VAR
	iter : FB_ObjCollectIterator;
END_VAR
//Bei dieser Methode wird der Node nur auf der Collection entnommen aber nicht gelöscht.
//Wird nur genutzt, wenn sich die Position eines Nodes im Object-Tree ändert (ExchangePiece)
IF pNode > 0 AND_THEN pNode^.nodes.nCount = 0 THEN
	M_GetIterator(iter);
	WHILE iter.pNode > 0 DO
		IF pNode = iter.pNode THEN
			IF pNode = pHead THEN
				pHead := pHead^.pNext;
				IF pHead > 0 THEN
					pHead^.pPrev := 0;	
				END_IF
			ELSIF pNode = pTail THEN
				pTail := pTail^.pPrev;
				IF pTail > 0 THEN
					pTail^.pNext := 0;	
				END_IF
			ELSE
				pNode^.pPrev^.pNext := pNode^.pNext;
				pNode^.pNext^.pPrev := pNode^.pPrev;
			END_IF
			pNode^.P_pOwnerColl := 0;
			nCount := nCount - 1;
			EXIT;
		END_IF
		iter.M_Increment();
	END_WHILE
END_IF
END_METHOD

END_FUNCTION_BLOCK

// ---- Configuration/FB_ObjCollectIterator.TcPOU
FUNCTION_BLOCK FB_ObjCollectIterator
VAR_INPUT
	pInitNode : POINTER TO FB_ObjCollectionNode;
END_VAR
VAR_OUTPUT
	pNode : POINTER TO FB_ObjCollectionNode;
END_VAR
VAR
END_VAR

pNode := pInitNode;

METHOD M_Increment
VAR_INPUT
END_VAR
IF pNode > 0 AND_THEN pNode^.pNext > 0 THEN
	pNode := pNode^.pNext;
ELSE
	pNode := 0;
END_IF
END_METHOD

END_FUNCTION_BLOCK

// ---- Configuration/FB_ObjCollectIteratorDeep.TcPOU
FUNCTION_BLOCK FB_ObjCollectIteratorDeep EXTENDS FB_ObjCollectIterator
VAR_INPUT
END_VAR
VAR_OUTPUT
END_VAR
VAR
	bBeforeInChild : BOOL;
	nLevel : UINT;
END_VAR

pNode := pInitNode;

METHOD M_Increment
VAR_INPUT
END_VAR

VAR
	
END_VAR
//Den kompletten Tree traversieren
//am Anfang steht der Iter auf dem Head von Level0
//wenn aktueller Node Childs hat, dann von diesen Childs neuen Iterator holen
//das geht immer so weiter bis ein Node keinen Child mehr hat
//wenn das eintritt, dann wird nach Nachbarn gesucht
//wenn ein Nachbar vorhanden, dann wird dieser zurückgegeben
//wenn kein Nachbar vorhanden, dann wird Parent zurückgegeben, hier besteht allerdings das Problem, dass
//wenn dann wieder inkrementiert wird, das Parent ja wieder auf das Child zugreifen würde. Ein Flag welches anzeigt,
//dass vorher schon in einer höheren Ebene dieses Parents gesucht wurde, könnte das lösen. Dieses muss allerdings immer
//an der richtigen stelle zurückgesetzt werden

IF pNode > 0 THEN
	IF pNode^.nodes.nCount > 0 THEN
		IF bBeforeInChild THEN
			//Nachbar suchen
			IF pNode^.pNext > 0 THEN
				pNode := pNode^.pNext;
			ELSE
				//kein Nachbar gefunden
				IF pNode^.pOwnerColl^.pOwnerNode > 0 THEN
					IF nLevel = 0 THEN
						pNode := 0;
						bBeforeInChild := FALSE;		
					ELSE
						//hier wird eine Ebene zurückgesprungen -> Flag setzen
						pNode := pNode^.pOwnerColl^.pOwnerNode;
						bBeforeInChild := TRUE;
						nLevel := nLevel - 1;
						THIS^.M_Increment();
					END_IF
				ELSE
					pNode := 0;
					bBeforeInChild := FALSE;		
				END_IF
			END_IF
			bBeforeInChild := FALSE;
		ELSE
			//Iterator vom neuen Child holen
			pNode^.nodes.M_GetIterator(THIS^);	//Hier wir das Level inkrementiert
			nLevel := nLevel + 1;
		END_IF
	ELSIF pNode^.pNext > 0 THEN
		//nach Nachbar suchen
		pNode := pNode^.pNext;
	ELSIF pNode^.pOwnerColl^.pOwnerNode > 0 AND nLevel > 0 THEN
		//hier wird eine Ebene zurückgesprungen -> Flag setzen
		pNode := pNode^.pOwnerColl^.pOwnerNode;
		bBeforeInChild := TRUE;
		nLevel := nLevel - 1;
		THIS^.M_Increment();
	ELSE
		pNode := 0;
		bBeforeInChild := FALSE;
	END_IF
END_IF
END_METHOD

END_FUNCTION_BLOCK

// ---- Objects/FB_Slot.TcPOU
{attribute 'enable_dynamic_creation'}
FUNCTION_BLOCK FB_Slot
VAR_INPUT
END_VAR
VAR_OUTPUT
END_VAR
VAR
	pOwner	: POINTER TO FB_Object;
	pChild	: POINTER TO FB_Object;
	nNr		: UINT;
	stRelPos: ST_3DPoint;
END_VAR

METHOD FB_init : BOOL
VAR_INPUT
	bInitRetains : BOOL; // if TRUE, the retain variables are initialized (warm start / cold start)
	bInCopyCode : BOOL;  // if TRUE, the instance afterwards gets moved into the copy code (online change)
	pOwner		: POINTER TO FB_Object;
END_VAR
THIS^.pOwner := pOwner;
END_METHOD

PROPERTY P_nNr : UINT
GET
P_nNr := nNr;
END_GET
SET
nNr := P_nNr;
END_SET
END_PROPERTY

PROPERTY P_rRelPosY : REAL
SET
stRelPos.Y := P_rRelPosY;
END_SET
GET
P_rRelPosY := stRelPos.Y;
END_GET
END_PROPERTY

PROPERTY P_rRelPosX : REAL
SET
stRelPos.X := P_rRelPosX;
END_SET
GET
P_rRelPosX := stRelPos.X;
END_GET
END_PROPERTY

PROPERTY P_pChild : POINTER TO FB_Object
GET
P_pChild := pChild;
END_GET
SET
pChild := P_pChild;
END_SET
END_PROPERTY

PROPERTY P_stRelPos : ST_3DPoint
SET
stRelPos := P_stRelPos;
END_SET
GET
P_stRelPos := stRelPos;
END_GET
END_PROPERTY

PROPERTY P_stAbsPos : ST_3DPoint
GET
VAR
	stTemp : ST_3DPoint;
	pMzTool: POINTER TO FB_MzTool;
	pTarget: POINTER TO FB_TargetBase;
END_VAR
IF pOwner^.P_eObjectType = E_ObjectType.OBJECTTYPE_MZHead THEN
	pMzTool := pOwner;
	stTemp := pMzTool^.P_stAbsPosTotal;
	stTemp.X := stTemp.X + stRelPos.X;
	stTemp.Y := stTemp.Y + stRelPos.Y;
	P_stAbsPos := stTemp;
ELSIF pOwner^.M_bIsGroup(E_ObjectGroup.OBJECTGROUP_MzTool) THEN
	pMzTool := pOwner;
	P_stAbsPos := F_Add3DPoints(stRelPos, pMzTool^.P_stAbsPosPhysExclPiece);
ELSIF pOwner^.M_bIsGroup(E_ObjectGroup.OBJECTGROUP_Target) THEN
	pTarget := pOwner;
	P_stAbsPos := F_Add3DPoints(stRelPos, pTarget^.P_stAbsPosLB);
END_IF
END_GET
END_PROPERTY

PROPERTY P_rRelPosZ : REAL
GET
P_rRelPosZ := stRelPos.Z;
END_GET
SET
stRelPos.Z := P_rRelPosZ;
END_SET
END_PROPERTY

END_FUNCTION_BLOCK

// ---- Objects/Tools/FB_MzTool.TcPOU
FUNCTION_BLOCK FB_MzTool EXTENDS FB_MzBase
VAR_INPUT
END_VAR
VAR_OUTPUT
END_VAR
VAR
	pParentMzTool		: POINTER TO FB_MzBase;
	
	nParentSlotNr		: UINT;	//LÖSCHEN!!!!!!!!!!!!!!!
	pZAxisRef 			: POINTER TO FB_ZAxisRef;
	pCurrentTarget		: POINTER TO FB_TargetBase;
	
	bIsMESTool			: BOOL;
	
	//Action: "JogZ"
	bJogZ				: BOOL;
	nStateA_JogZ		: USINT;			//State von A_Jog()
	fbZmJog				: FB_ZM_Jog;
	eJogZDirectionNew	: E_MoveDirection;
	eJogZDirection		: E_MoveDirection;
	bJogZForward		: BOOL;
	bJogZBackwards		: BOOL;
	bJogZClock			: BOOL;
	bJogZModeInchingNew	: BOOL;				//wenn True dann Tipbetrieb sonst kontinuierlich
	bJogZModeInching	: BOOL;				//wenn True dann Tipbetrieb sonst kontinuierlich
	rJogZDistance		: REAL;
	rJogZSpeed			: REAL;
	bJogZImpuls			: BOOL;
	
	//Ergänzung zu Action: MoveZ"
	nReducedMoveZSpeed	: DINT;
	nReducedMoveZDist	: DINT;
	
END_VAR

IF eCurrentState = E_MachineState.MACHINESTATE_Active THEN
	//BasicActions ausführen
	IF bJogZ THEN
		A_JogZ();
		IF nStateA_JogZ >= 80 THEN
			IF nStateA_JogZ >= 99 THEN
				bStopAllOnError := TRUE;
				bError := TRUE;
			END_IF
		bJogZ := FALSE;
		nStateA_JogZ := 0; 
		M_RemoveListEntry(nSearchValue:= E_Action.ACTION_Jog);
		END_IF
	END_IF
END_IF


SUPER^();	//FB_MzBase() aufrufen

//Prozessdaten aktualisieren
IF pZAxisRef > 0 THEN
	stProcessData.n32Data[3] := REAL_TO_DINT(pZAxisRef^.P_rCurrentPos);
END_IF
stCurrentPos := P_stCurrentPosTotal;
stProcessData.n32Data[4] := REAL_TO_DINT(stCurrentPos.X);
stProcessData.n32Data[5] := REAL_TO_DINT(stCurrentPos.Y);
stProcessData.n32Data[6] := REAL_TO_DINT(stCurrentPos.Z);

ACTION A_Init:
	IF nStateA_InitAxis = 0 THEN
		bInitAxisOk := FALSE;
		//Ist Z-Achse physikalisch vorhanden?
		IF NOT pZAxisRef^.stInput.nStatus.7 THEN
			stError.ErrorId := E_ErrorIdMultiZ.ERRORID_NoZAxis;
			stError.HardwareGrp := E_HardwareGrp.AxisZ;
			stError.HardwareNr	:= pZAxisRef^.nChannel;
			stError.POUState := nStateA_InitAxis;
			nStateA_InitAxis := 99;
		ELSE
			IF pZAxisRef^.stStatus.bIsHoming THEN //Homing dieser Achse wurde bereits durch ein anderes Tool oder Head angestoßen
				nStateA_InitAxis := 2;
			ELSE
				nStateA_InitAxis := 1;
			END_IF		
		END_IF
	END_IF
	
	IF nStateA_InitAxis = 1 THEN
		fbZmHome(bExecute:= TRUE, pFbZAxisRef:= pZAxisRef, bMoveToHome:= TRUE);
		P_bZIsMoving := TRUE;
		pParentMzTool^.P_bZIsMoving := TRUE;		
		IF NOT fbZmHome.bBusy THEN
			IF fbZmHome.bError THEN
				stError.ErrorId := fbZmHome.nErrorId;
				stError.HardwareGrp := E_HardwareGrp.AxisZ;
				stError.HardwareNr	:= pZAxisRef^.nChannel;
				stError.POUState := nStateA_InitAxis;
				nStateA_InitAxis := 99;
			ELSE
				bInitAxisOk := TRUE;
				nStateA_InitAxis := 80;
			END_IF
			fbZmHome(bExecute:= FALSE);
			pParentMzTool^.P_bZIsMoving := FALSE;
			P_bZIsMoving := FALSE;
		END_IF			
	END_IF
	
	//Achse wurde durch anderes Tool angestoßen -> warten bis Homing fertig
	IF nStateA_InitAxis = 2 THEN
		IF NOT pZAxisRef^.stStatus.bIsHoming THEN
			IF pZAxisRef^.stStatus.bError THEN
				nStateA_InitAxis := 99;
			ELSIF pZAxisRef^.stStatus.bCmdAborted THEN
				nStateA_InitAxis := 80;	
			ELSIF pZAxisRef^.stStatus.bIsHomed THEN
				bInitAxisOk := TRUE;
				nStateA_InitAxis := 80;
			END_IF
		END_IF
	END_IF

	IF nStateA_InitAxis = 70 THEN
		pParentMzTool^.P_bZIsMoving := FALSE;
		P_bZIsMoving := FALSE;
		fbZmHome(bExecute:= FALSE);
		nStateA_InitAxis := 80;
	END_IF

//Errorhandling
IF nStateA_InitAxis = 99 THEN
	stError.ObjectId := nObjectID;
	stError.Cmd := E_Action.ACTION_Init;
	stError.POU := E_POU.POU_FB_MzTool;
	stError.POUAction := E_POUACT.POUACT_A_Init;
	fbErrorList.M_Add(stError);
END_IF
END_ACTION

ACTION A_JogZ:
IF nStateA_JogZ = 0 THEN
	IF bJogZModeInching THEN
		nStateA_JogZ := 1;	//Incr
	ELSE
		nStateA_JogZ := 3;	//Continous
	END_IF
END_IF
 
IF nStateA_JogZ = 1 THEN	//incrementellen Jog-Befehl 1x absetzen
	CASE eJogZDirection OF
		E_MoveDirection.DIRECTION_ZPLUS:
			IF pZAxisRef > 0 THEN
				fbZmJog(bJogForward:= TRUE, bJogBackwards:= FALSE, bClock:= bJogZClock, bInching:= TRUE,
						rSpeed:= rJogZSpeed, rDistance:= rJogZDistance, pfbZAxisRef:= pZAxisRef);					
			END_IF
			bZIsMoving := TRUE;
		E_MoveDirection.DIRECTION_ZMINUS:
			IF pZAxisRef > 0 THEN
				fbZmJog(bJogForward:= FALSE, bJogBackwards:= TRUE, bClock:= bJogZClock, bInching:= TRUE,
						rSpeed:= rJogZSpeed, rDistance:= rJogZDistance, pfbZAxisRef:= pZAxisRef);					
			END_IF
			bZIsMoving := TRUE;		
	END_CASE
	nStateA_JogZ := 2;
END_IF

IF nStateA_JogZ = 2 THEN //warten bis inkrementelles Joggen fertig bzw auf neuen Befehl warten
	IF NOT bJogZModeInching THEN //Wechseln zu kontinulierlichem Joggen
		nStateA_JogZ := 3;
	END_IF
	
	IF eJogZDirection = E_MoveDirection.DIRECTION_STOP THEN
		nStateA_JogZ := 4;
	END_IF
END_IF

IF nStateA_JogZ = 3 THEN //zyclisches Absetzen des kontinuierlichen Jog-Befehls, hier kann auch Stop abgesetzt werden, bzw neuer inkr. Befehl
	IF bJogZImpuls THEN
		CASE eJogZDirection OF
			E_MoveDirection.DIRECTION_STOP:
				nStateA_JogZ := 4;
			E_MoveDirection.DIRECTION_ZPLUS:
				IF pZAxisRef > 0 THEN
					fbZmJog(bJogForward:= TRUE, bJogBackwards:= FALSE, bClock:= bJogZClock, bInching:= FALSE,
							rSpeed:= rJogZSpeed, rDistance:= rJogZDistance, pfbZAxisRef:= pZAxisRef);						
				END_IF
				bZIsMoving := TRUE;
			E_MoveDirection.DIRECTION_ZMINUS:
				IF pZAxisRef > 0 THEN
					fbZmJog(bJogForward:= FALSE, bJogBackwards:= TRUE, bClock:= bJogZClock, bInching:= FALSE,
							rSpeed:= rJogZSpeed, rDistance:= rJogZDistance, pfbZAxisRef:= pZAxisRef);					
				END_IF
				bZIsMoving := TRUE;	
		END_CASE
	END_IF
	bJogZImpuls := FALSE;
END_IF

IF nStateA_JogZ = 4 THEN //STOP
	IF fbZmJog.bBusy THEN
		fbZmJog(bJogForward:= FALSE, bJogBackwards:= FALSE, pfbZAxisRef:= pZAxisRef);
	END_IF
	nStateA_JogZ := 5;
END_IF

//Abfragen, ob Jogging fertig
fbZmJog(pfbZAxisRef:= pZAxisRef);
IF NOT fbZmJog.bBusy THEN
	nStateA_JogZ := 80;
	IF fbZmJog.bError THEN
		stError.Cmd := E_Action.ACTION_Jog;
		stError.ErrorId := fbZmJog.nErrorID;
		stError.HardwareGrp := E_HardwareGrp.AxisZ;
		stError.HardwareNr	:= pZAxisRef^.nChannel;
		stError.POU := E_POU.POU_FB_MzTool;
		stError.POUAction := E_POUACT.POUACT_A_JogZ;
		stError.POUState := nStateA_JogZ;
		fbErrorList.M_Add(stError);
		nStateA_JogZ := 99;
		fbZmJog.M_Reset();
	END_IF
	bZIsMoving := FALSE;
END_IF
END_ACTION

ACTION A_MoveZ:
CASE nStateA_MoveZ OF
	0:
	IF bFlagMoveZ THEN
		//Wenn Achse von einem anderen Tool bereits Fahrauftrag, dann warten bis dieser abgearbeitet
		IF pZAxisRef^.stStatus.bHasJob THEN
			RETURN;
		END_IF

		fbZmMove.eMoveMode := eMoveModeZ;
		fbZmMove.rSpeed := rMoveSpeedZ;
		fbZmMove.rPosition := rMovePositionZ;
		
		CASE eMoveModeZ OF
			E_MoveMode.MODE_AbsWithOffset:
				//TargetPosition in Achsenposition umgerechnen
				//Die Targetposition der ZAchse ergibt sich: AxisPosZ = TargetPosZ - AbsPos.Z
				//zu beachten ist, dass sich Bedeutung von AbsPos.Z zu AbsPos.X und AbsPos.Y unterscheidet (siehe Property P_AbsPos)
				st3DPoint := P_stAbsPosTotal;
				fbZmMove.rPosition := rMovePositionZ - st3DPoint.Z;
				
			E_MoveMode.MODE_Free:
				//aus dem kollisionsgefährdetem Bereich herausfahren
				st3DPoint := P_stCurrentPosPhys;
				IF st3DPoint.Z >= pAssignWorkplate^.P_rCollHeight THEN //ist bereits außerhalb des Bereichs
					nStateA_MoveZ := 80;
					RETURN;
				END_IF
				
				IF nReducedMoveZSpeed > 0 THEN //Zuerst einen Move relativ um nReducedMoveZDistance
					fbZmMove.eMoveMode := E_MoveMode.MODE_Relative;
					fbZmMove.rPosition := DINT_TO_REAL(nReducedMoveZDist);
					fbZmMove.rSpeed := DINT_TO_REAL(nReducedMoveZSpeed);
				ELSE
					//TargetPosition in Achsenposition umgerechnen
					//Die Targetposition der ZAchse ergibt sich: AxisPosZ = TargetPosZ - AbsPos.Z
					//zu beachten ist, dass sich Bedeutung von AbsPos.Z zu AbsPos.X und AbsPos.Y unterscheidet (siehe Property P_AbsPos)
					//st3DPoint := P_stAbsPosTotal;	//Summe aller Offsets
					st3DPoint := P_stAbsPosPhys;
					fbZmMove.rPosition := pAssignWorkplate^.P_rCollHeight - st3DPoint.Z;
				END_IF				
				
				stAreaCollFree.M_Clear();
			E_MoveMode.MODE_Home:	
				//bei "Home wird vorerst keine Position übergeben, nur bei unterem Kopf?
				IF nReducedMoveZSpeed > 0 THEN //Zuerst einen Move relativ um nReducedMoveZDistance
					fbZmMove.eMoveMode := E_MoveMode.MODE_Relative;
					fbZmMove.rPosition := DINT_TO_REAL(nReducedMoveZDist);
					fbZmMove.rSpeed := DINT_TO_REAL(nReducedMoveZSpeed);
				END_IF				
				stAreaCollFree.M_Clear();
		END_CASE
	END_IF
	
	IF bFlagMoveZ XOR fbZmMove.bBusy THEN
		bFlagMoveZ := FALSE;
		fbZmMove(bExecute:= TRUE, pfbZAxisRef:= pZAxisRef);
	END_IF 

	IF NOT fbZmMove.bBusy THEN
		IF fbZmMove.bError THEN
			stError.ErrorId := fbZmMove.nErrorID;
			stError.Cmd := E_Action.ACTION_MoveZ;
			stError.HardwareGrp := E_HardwareGrp.AxisZ;
			stError.HardwareNr	:= pZAxisRef^.nChannel;
			stAreaCollFree.M_Clear();
			stError.POUState := nStateA_MoveZ;					 
			nStateA_MoveZ := 99;
		ELSE
			st3DPoint := P_stCurrentPosTotal;
			stAreaCollFree.X1 := st3DPoint.X - stAreaCollFree.X1;
			stAreaCollFree.X2 := st3DPoint.X + stAreaCollFree.X2;
			stAreaCollFree.Y1 := st3DPoint.Y - stAreaCollFree.Y1;
			stAreaCollFree.Y2 := st3DPoint.Y + stAreaCollFree.Y2;
			IF (eMoveModeZ = E_MoveMode.MODE_Free  OR eMoveModeZ = E_MoveMode.MODE_Home) AND nReducedMoveZSpeed > 0 THEN
				nReducedMoveZSpeed := 0;
				nReducedMoveZDist := 0;
				nStateA_MoveZ := 0;
			ELSE
				nStateA_MoveZ := 80;
			END_IF
		END_IF
		fbZmMove(bExecute:= FALSE);
		bFlagMoveZ := TRUE;
	END_IF			
	
	70:	//Stoppen
		fbZmStop(pFbZAxisRef:= pZAxisRef, bExecute:= TRUE);
		IF NOT fbZmStop.bBusy THEN
			IF fbZmStop.bError THEN
				stError.Cmd := E_Action.ACTION_Stop;
				stError.ErrorId := fbZmStop.nErrorID;
				stError.HardwareGrp := E_HardwareGrp.AxisZ;
				stError.HardwareNr	:= pZAxisRef^.nChannel;
				stError.POUState := nStateA_MoveZ;
				nStateA_MoveZ := 99;
			ELSE
				nStateA_MoveZ := 80;
				nReducedMoveZSpeed := 0;
				nReducedMoveZDist := 0;
			END_IF
			fbZmMove(bExecute:= FALSE,pfbZAxisRef:= pZAxisRef);
			fbZmStop(bExecute:= FALSE,pfbZAxisRef:= pZAxisRef);
			bFlagMoveZ := TRUE;
			stAreaCollFree.M_Clear();
		END_IF;
END_CASE

//Errorhandling
IF nStateA_MoveZ = 99 THEN
	stError.ObjectId := nObjectID;
	stError.POU := E_POU.POU_FB_MzTool;
	stError.POUAction := E_POUACT.POUACT_A_MoveZ;
	fbErrorList.M_Add(stError);
END_IF
END_ACTION

ACTION A_Reset:
IF bJogZ THEN
	bJogZ := FALSE;
	nStateA_JogZ := 0;
END_IF		

IF nStateA_ResetTool = 0 THEN
	//Warten, bis Axis wieder fehlerfrei
	IF NOT pFbMultiZ^.bBusy THEN
		IF NOT pZAxisRef^.stStatus.bError THEN
			nStateA_ResetTool := 1;				
		END_IF
	END_IF
END_IF

IF nStateA_ResetTool = 1 THEN
	IF nStateA_ResetSpec = 80 THEN
		nStateA_ResetTool := 80;
	END_IF
END_IF

SUPER^.A_Reset();
END_ACTION

ACTION A_Stop:
//Diese Aktion wird in der Regel vom "FB_Spec.A_stop()" aufgerufen
//kommt der Aufruf von "FB_Spec.A_stop()" das erste mal, ist "nStateA_Stop" = 1

//Abgebrochen werden muss "JogZ" und "MoveZ" 
IF nStateA_Stop <= 1 THEN
	IF bJogZ AND nStateA_JogZ < 4 THEN
		nStateA_JogZ := 4;
	END_IF

	nStateA_Stop := 2;
END_IF

SUPER^.A_Stop();
END_ACTION

METHOD M_AddChild : ERRORID
VAR_INPUT
	pObject : POINTER TO FB_Object;
	nSlotNr	: UINT;
	nIndex : INT;
END_VAR

VAR
	pSlot : POINTER TO FB_Slot;
END_VAR
//In den abgeleiteten Tool-FBs wird überprüft, ob das entsprechende Objekt als Child geeignet ist
IF pObject > 0 THEN
	pSlot := fbSlotList.M_GetAtNr(nSlotNr);
	IF pSlot > 0 THEN
		IF pSlot^.P_pChild = 0 THEN
			//Object darf selber noch an keinem Parent hängen
			IF pObject^.P_pParentObject = 0 THEN
				pSlot^.P_pChild := pObject;
				IF pObject^.M_bIsGroup(E_ObjectGroup.OBJECTGROUP_Piece) THEN
					//Piece gehört immer an den letzten Slot
					IF pSlot^.P_nNr = nNumberOfSlots THEN
						pPiece := pObject;
					ELSE
						M_AddChild := E_ErrorIdObjMgmt.ERRORID_InvalidSlotNumber;
						RETURN;
					END_IF
				END_IF
 				pObject^.P_pObjCollectNode := pObjCollectNode^.nodes.M_AddNewNode(pObject,nIndex);
				pObject^.M_UpdateParent();
			ELSE
				M_AddChild := E_ErrorIdObjMgmt.ERRORID_ObjectAlreadyOnAnotherParent;
			END_IF
		ELSE //Slot bereits belegt
			M_AddChild := E_ErrorIdObjMgmt.ERRORID_SlotIsAlreadyOccupied;
		END_IF		
	ELSE
		M_AddChild := E_ErrorIdObjMgmt.ERRORID_InvalidSlotNumber;			
	END_IF
ELSE
	M_AddChild := E_ErrorIdObjMgmt.ERRORID_InvalidParentObject;
END_IF
END_METHOD

METHOD M_AnswerSiblingForAction : ERRORID
VAR_INPUT
	eAction : E_Action;
END_VAR
END_METHOD

METHOD M_AskSiblingForAction : ERRORID
VAR_INPUT
	eAction : E_Action;
END_VAR

VAR
	iter : FB_ObjCollectIteratorDeep;
	pTool : POINTER TO FB_MzTool;
END_VAR
//Mit dieser Methode wird überprüft, ob ein an dieser Achse hängendes anderes Tool ein spezielle Methode
//für dieses Tool verhindert. Z.B. wird dadurch verhindert, dass eine einzelne Pipette am TitrationsTool
//einen MoveToTarget ausführt, obwohl am TitrationsTool ein Cap steckt.

//Das Tool ermitteln, welches an der Achse selber hängt, denn dort kann nur eines hängen
P_pUpperParentTool^.P_pObjCollectNode^.nodes.M_GetIterator(iter);
WHILE iter.pNode > 0 DO
	IF iter.pNode^.P_pObject > 0 AND_THEN iter.pNode^.P_pObject^.M_bIsGroup(E_ObjectGroup.OBJECTGROUP_MzTool) THEN
		pTool := iter.pNode^.P_pObject;
		IF pTool <> THIS THEN
			M_AskSiblingForAction := pTool^.M_AnswerSiblingForAction(eAction);
			IF M_AskSiblingForAction > 0 THEN
				RETURN;
			END_IF
		END_IF
	END_IF
	iter.M_Increment();	
END_WHILE
END_METHOD

METHOD M_CancelAction
VAR_INPUT
	eAction : E_Action;
END_VAR
IF eAction = E_Action.ACTION_MoveZ THEN
	IF bMoveZ AND nStateA_MoveZ < 70 THEN
		nStateA_MoveZ := 70;
	END_IF
ELSIF eAction = E_Action.ACTION_Jog THEN
	IF bJogZ AND nStateA_JogZ < 4 THEN
		nStateA_JogZ := 4;
	ELSE
		SUPER^.M_CancelAction(eAction);	
	END_IF
ELSE
	SUPER^.M_CancelAction(eAction);
END_IF
END_METHOD

METHOD M_CheckAction : ERRORID
VAR_INPUT
	refActionData 	: REFERENCE TO ST_ActionData;
	pCorrelObject	: POINTER TO FB_Object;
END_VAR
//abgeleiteten Klassen separat eingeschränkt
IF refActionData.eAction = E_Action.ACTION_MoveToTarget THEN
	//MoveToTarget darf nicht aufgeführt werden, wenn Tool ChildTools besitzt und diese
	//näher zur Worlplate sind (bsp. CartrideHolder und CartridgeDispenser)
	IF M_GetClosestTool(bAllOnAxis:= FALSE) <> THIS THEN
		M_CheckAction := E_ErrorIdCmd.ERRORID_ActionLocked;
	END_IF
ELSIF refActionData.eAction = E_Action.ACTION_ActionOnArray THEN
	RETURN;
ELSE
	M_CheckAction := SUPER^.M_CheckAction(refActionData,pCorrelObject);
END_IF
END_METHOD

METHOD M_CheckMoveLimit : BOOL
VAR_INPUT
	sAxis			: STRING[2];
	eMoveMode		: E_MoveMode;
	rMovePosition	: REAL;
END_VAR

VAR
	st3DPoint		: ST_3DPoint;
	rMovePosTemp	: REAL;
END_VAR
IF sAxis = 'Z' THEN 
	IF eMoveMode = E_MoveMode.MODE_Relative OR eMoveMode = E_MoveMode.MODE_Measure THEN	//Relativ
		rMovePosTemp := pZAxisRef^.P_rCurrentPos + rMovePosition;
	ELSIF eMoveMode = E_MoveMode.MODE_AbsWithOffset THEN	//Absolut mit Offsets
		st3DPoint := P_stAbsPosTotal;	//Summe aller Offsets
		rMovePosTemp :=  rMovePosition - st3DPoint.Z;
	ELSIF eMoveMode = E_MoveMode.MODE_AbsNoneOffset THEN	//Absolut OHNE Offsets!!
		rMovePosTemp := rMovePosition;
	ELSIF eMoveMode = E_MoveMode.MODE_Free OR eMoveMode = E_MoveMode.MODE_Home THEN	//Free
		M_CheckMoveLimit := TRUE;
	END_IF
	
	IF rMovePosTemp >= pZAxisRef^.P_rMinPos AND rMovePosTemp <= pZAxisRef^.P_rMaxPos THEN
		M_CheckMoveLimit := TRUE;
	END_IF
ELSE
	M_CheckMoveLimit := SUPER^.M_CheckMoveLimit(sAxis,eMoveMode,rMovePosition);
END_IF
END_METHOD

METHOD M_CheckMoveLimitEx : ERRORID
VAR_INPUT
	LimitCuboid : REFERENCE TO FB_Cuboid;
END_VAR

VAR
	stAbsPosTotal : ST_3DPoint;
END_VAR
stAbsPosTotal := P_stAbsPosTotal;

IF LimitCuboid.P_rXMin < pXDrive^.P_rMinPos + stAbsPosTotal.X OR LimitCuboid.P_rXMax > pXDrive^.P_rMaxPos + stAbsPosTotal.X THEN
	M_CheckMoveLimitEx := E_ErrorIdGCode.ERRORID_ScaffoldWidthExceeded; 
END_IF

IF LimitCuboid.P_rYMin < pYDrive^.P_rMinPos + stAbsPosTotal.Y OR LimitCuboid.P_rYMax > pYDrive^.P_rMaxPos + stAbsPosTotal.Y THEN
	M_CheckMoveLimitEx := E_ErrorIdGCode.ERRORID_ScaffoldDepthExceeded;
END_IF

IF LimitCuboid.P_rZMin < pZAxisRef^.P_rMinPos + stAbsPosTotal.Z OR LimitCuboid.P_rZMax > pZAxisRef^.P_rMaxPos + stAbsPosTotal.Z THEN
	M_CheckMoveLimitEx := E_ErrorIdGCode.ERRORID_ScaffoldHeightExceeded;
END_IF
END_METHOD

METHOD M_CheckProps : ERRORID
VAR_INPUT
END_VAR
M_CheckProps := SUPER^.M_CheckProps();
pAssignWorkplate := pParentMzTool^.P_pAssignWorkplate;
IF pZAxisRef = 0 THEN
	M_CheckProps := E_ErrorIdObjMgmt.ERRORID_InvalidParentMzTool;
END_IF
END_METHOD

METHOD M_ClearAllProps
VAR_INPUT
	bIgnoreParent : BOOL; //Es wird das gesamte OD gelöscht. -> Zeiger auf Parent nicht mehr gültig!
END_VAR
VAR
	pSlot : POINTER TO FB_Slot;
END_VAR
//Vom Parent lösen, falls dieses noch existiert
IF NOT bIgnoreParent AND_THEN pParentMzTool > 0 THEN
	pSlot := pParentMzTool^.M_GetSlotFromChild(THIS); 
	IF pSlot > 0 THEN
		IF pSlot^.P_pChild^.P_nObjectID = nObjectID THEN
			pSlot^.P_pChild := 0;
		END_IF
	END_IF
END_IF

pParentMzTool := 0;

IF pZAxisRef > 0 THEN
	pZAxisRef^.eFixedToolType := E_MzToolType.TOOL_TYPE_None;
END_IF

SUPER^.M_ClearAllProps(bIgnoreParent);
END_METHOD

METHOD M_ExeAction : ERRORID
VAR_INPUT
	refActionData : REFERENCE TO ST_ActionData;	
END_VAR

VAR
	rAbsFreeHeight : REAL; 
END_VAR
//In dieser Methode muss gecheckt werden, ob die entsprechende BasicAction auch zum aktuellen Zeitpunkt auch ausgeführt werden kann
bCanceled := FALSE;

IF NOT (eCurrentState = E_MachineState.MACHINESTATE_Idle OR
	eCurrentState = E_MachineState.MACHINESTATE_Active OR
	eCurrentState = E_MachineState.MACHINESTATE_Ready) THEN
	M_ExeAction := E_ErrorIdCmd.ERRORID_InvalidState;
	RETURN;
END_IF

CASE refActionData.eAction OF
	E_Action.ACTION_Init:
		IF NOT bInitAxis THEN
			bReInit := DINT_TO_BOOL(refActionData.aParams[1]);
			bInitAxis := TRUE;			
			fbList.A_AddHeadValue(hList := hList, putValue := E_Action.ACTION_Init); 
			//bIsInit := FALSE;
		ELSE
			RETURN;
		END_IF
		
	E_Action.ACTION_Jog:
		//Action darf eingetragen werden wenn:
		//wenn Action noch nicht aktiv oder
		//wenn Action aktiv und nJogDirection = 0
		//wenn Action aktiv und Jogmode = Continous und aktueller Jogmode = Continous
		
		//Wenn X ode Y dann auf FB_MzBase verweisen

		eJogZDirectionNew := DINT_TO_USINT(refActionData.aParams[2]);
		bJogZModeInchingNew := DINT_TO_BOOL(refActionData.aParams[1]);
		
		//Speed auf max Axisspeed begrenzen
		rJogZSpeed := MIN(DINT_TO_REAL(refActionData.aParams[3]),pZAxisRef^.P_rMaxSpeed);
		rJogZDistance := DINT_TO_REAL(refActionData.aParams[4]);
		
		IF eJogZDirectionNew < 5 THEN //X,Y oder Stop
			M_ExeAction := SUPER^.M_ExeAction(refActionData);
			IF 	eJogZDirectionNew > 0 THEN
				RETURN;
			END_IF
		END_IF

		//Wenn es einen Richtungswechsel gibt, dann darf "bJog" nicht aktiv sein
		IF NOT bJogZ THEN 
			IF eJogZDirectionNew  = E_MoveDirection.DIRECTION_ZMINUS THEN //Z nach unten
				//ermitteln, über welchem Target sich MzTool befindet und die maximale Joggingdistanz ermitteln
				{warning 'Noch implementieren'}
				//Aufgabe für später: hängen an einer Achse mehrere MzTools, dann muss das für diese auch ermittelt werden
				IF rJogZSpeed > 5000.0 THEN
					pCurrentTarget := pAssignWorkplate^.M_GetHighestTarget(P_stCurrentXYArea,0);
					//nJogDistance aus TargetPosition Z umrechnen in Raw-Position
					MEMSET(ADR(st3DPoint1),0,SIZEOF(st3DPoint1));
					IF pCurrentTarget > 0 THEN
						rAbsFreeHeight := pCurrentTarget^.P_rAbsFreeHeight;
					ELSE
						RETURN;
					END_IF
					
					IF bJogZModeInchingNew THEN
						//st3DPoint := P_stCurrentPosPhys;
						st3DPoint := M_GetClosestTool(bAllOnAxis:= TRUE)^.P_stCurrentPosPhys;
						//nJogDistance reduzieren, so dass nicht aufsetzt
						//aktuelle Position
						IF P_pMzHead^.P_bIsTopHead THEN	//oberhalb der Workplate
							IF st3DPoint.Z <= rAbsFreeHeight + 3000.0 THEN
								RETURN;
							END_IF
							rJogZDistance := MIN(st3DPoint.Z - rAbsFreeHeight - 3000.0, rJogZDistance);
						END_IF
 					ELSE //Continous
						IF P_pMzHead^.P_bIsTopHead THEN	//oberhalb der Workplate
							//Fall das Target im Weg, dann die JogDistance berechnen und Sicherheitsabstand abziehen
							//st3DPoint := P_stCurrentPosPhys;
							st3DPoint := M_GetClosestTool(bAllOnAxis:= TRUE)^.P_stCurrentPosPhys;
							rJogZDistance := MAX(st3DPoint.Z - rAbsFreeHeight -3000.0,0.0);
						ELSE
							rJogZDistance := 999999.9;	
						END_IF
					END_IF
				ELSE
					IF NOT bJogZModeInchingNew THEN
						rJogZDistance := 999999.9;
					END_IF
				END_IF
			ELSE
				IF NOT bJogZModeInchingNew THEN
					rJogZDistance := 999999.9;
				END_IF
			END_IF
		END_IF
		
		IF bJogZ THEN	//Aktion schon akiv
			//nJogDirection = 0 oder bleibt oder neuer und alter JogMode = Continous
			IF NOT ((eJogZDirectionNew = E_MoveDirection.DIRECTION_STOP) OR 
					((eJogZDirectionNew = eJogZDirection) AND
					(bJogZModeInchingNew = FALSE AND bJogZModeInching = FALSE))) THEN
				RETURN;
			END_IF
 		END_IF
	
		eJogZDirection := eJogZDirectionNew;
		bJogZModeInching := bJogZModeInchingNew;
		
		//In LinkedListCtrl eintragen - wenn schon vorhanden, dann überschreiben!!
		getPosPtr := 0;	//nach vorhandenem Eintrag suchen - beginnen an Anfang
		fbList.A_FindNext(hList := hList, putPosPtr := getPosPtr, putValue := E_Action.ACTION_Jog, getValue=>getValue, getPosPtr=>getPosPtr );

		IF NOT fbList.bOk THEN	//Eintrag wurde nicht gefunden
			//Übeprüfen, ob Achse referenziert
			 IF NOT pZAxisRef^.stStatus.bIsHomed THEN
				M_ExeAction := E_ErrorIdMultiZ.ERRORID_AxisNotHomed;
				RETURN;
			 END_IF
			bJogZ := TRUE;
			bJogZImpuls := TRUE;
			bJogZClock := TRUE;			
			fbList.A_AddHeadValue(hList := hList, putValue := E_Action.ACTION_Jog);
			bBusy := TRUE;
		ELSE	//Eintrag wurde gefunden
			bJogZClock := NOT bJogZClock;
			bJogZImpuls := TRUE;
		END_IF
	
	E_Action.ACTION_MoveZ:
		IF NOT bMoveZ THEN
			//Checken, ob Achse initialisiert
			IF NOT P_bIsInit THEN
				M_ExeAction := E_ErrorIdCmd.ERRORID_DeviceNotInitialized;
				RETURN;
			END_IF
			
			//Check MoveMode nicht notwendig, da für Z alle zulässig sind
			eMoveModeZ := DINT_TO_USINT(refActionData.aParams[1]);
			
			IF eMoveModeZ = E_MoveMode.MODE_Free AND bDisableFreeMove THEN
				bDisableFreeMove := FALSE;
				RETURN;
			END_IF
			
			bDisableFreeMove := FALSE;
			
			//Action darf nicht ausgeführt werden wenn:
			IF eObjectType = E_ObjectType.OBJECTTYPE_MZHead THEN
				//Head darf nur alle in ihm hängende Tools freifahren oder auf "0" fahren
				IF eMoveModeZ = E_MoveMode.MODE_Free OR eMoveModeZ = E_MoveMode.MODE_Home THEN
					bMoveZ := TRUE;			
					fbList.A_AddHeadValue(hList := hList, putValue := E_Action.ACTION_MoveZ);
				ELSE
					M_ExeAction := E_ErrorIdObjMgmt.ERRORID_IsNoMzTool;
					RETURN;
				END_IF
			ELSE
				IF bZIsMoving THEN	//Z-Achse selber schon in Bewegung
					M_ExeAction := E_ErrorIdMultiZ.ERRORID_MultiZIsStillMoving;
					RETURN;
				ELSIF pParentMzTool^.P_bXYIsMoving THEN	//Kopf ist in XY schon in Bewegung (hier sind allerding die Home und Free Modi erlaubt)
					IF NOT (eMoveModeZ = E_MoveMode.MODE_Free OR eMoveModeZ = E_MoveMode.MODE_Home) THEN
						M_ExeAction := E_ErrorIdMultiZ.ERRORID_MultiZIsStillMoving;
						RETURN;
					END_IF
				ELSIF NOT pZAxisRef^.stStatus.bIsHomed THEN //sie nicht referenziert ist
					M_ExeAction := E_ErrorIdMultiZ.ERRORID_AxisNotHomed;
					RETURN;
				END_IF
				
				rMovePositionZ := DINT_TO_REAL(refActionData.aParams[2]);
				
				//"E_MoveMode.MODE_Measure" nur für ZSensor zulässig
				IF eMoveModeZ = E_MoveMode.MODE_Measure THEN
				  IF eObjectType = E_ObjectType.OBJECTTYPE_ZSensor THEN
					 //Im Mode "Measure" ist die MovePos negativ (Vermessung nach unten)
					 //falls die MovePos außerhalb der Erreichbarkeit der Achse liegt, dann auf MinPos beschränken
					 //ist notwendig, da der ZSensor zum Vermessen etwas tiefer fahren muss als das Target liegt
					 //und bei Targets, die geradeso erreichbar wären, ein Limit-Error auftreten würde
					 //siehe ToDo #465
					 rMovePositionZ := MAX((pZAxisRef^.P_rMinPos - pZAxisRef^.P_rCurrentPos),rMovePositionZ);
				  ELSE
					M_ExeAction := E_ErrorIdCmd.ERRORID_InvalidMoveMode;
					RETURN;
				  END_IF
				END_IF
	
				//Position auf Limits checken
				IF NOT M_CheckMoveLimit(sAxis:= 'Z', eMoveMode:= eMoveModeZ,rMovePosition:= rMovePositionZ) THEN
					M_ExeAction := E_ErrorIdCmd.ERRORID_TargetPosOutOfRangeZ;
					RETURN;
				END_IF
				
				rMoveSpeedZ := MIN(DINT_TO_REAL(refActionData.aParams[3]),pZAxisRef^.P_rMaxSpeed);
				
				 //Geschwindigkeitsangabe -1 = max. Geschwindigkeit
				IF rMoveSpeedZ < 0 OR eMoveModeZ = E_MoveMode.MODE_Home OR eMoveModeZ = E_MoveMode.MODE_Free THEN
					rMoveSpeedZ := pZAxisRef^.P_rMaxSpeed;
				END_IF
				
				stAreaCollFree.X1 := DINT_TO_REAL(refActionData.aParams[4]);
				stAreaCollFree.X2 := DINT_TO_REAL(refActionData.aParams[5]);
				stAreaCollFree.Y1 := DINT_TO_REAL(refActionData.aParams[6]);
				stAreaCollFree.Y2 := DINT_TO_REAL(refActionData.aParams[7]);
				
				bZIsMoving := TRUE;
				bMoveZ := TRUE;			
				fbList.A_AddHeadValue(hList := hList, putValue := E_Action.ACTION_MoveZ);
			END_IF
		ELSE
			M_ExeAction := E_ErrorIdCmd.ERRORID_BasicActionActive;  //Error
			RETURN;				
		END_IF
	ELSE
		M_ExeAction := SUPER^.M_ExeAction(refActionData);
		RETURN;;
END_CASE

eCurrentState := E_MachineState.MACHINESTATE_Active;
bBusy := TRUE;
END_METHOD

METHOD M_GetAllProps : ERRORID
VAR_INPUT
	refCmdData : REFERENCE TO  ST_CmdData;
END_VAR
//Basisproperties lesen
SUPER^.M_GetAllProps(refCmdData);

refCmdData.n32Data[0] := pParentMzTool^.P_nObjectID;

IF pParentSlot > 0 THEN
	refCmdData.n32Data[1] := pParentSlot^.P_nNr;
ELSE
	refCmdData.n32Data[1] := 0;
END_IF
END_METHOD

METHOD M_GetClosestTool : POINTER TO FB_MzTool
VAR_INPUT
	bAllOnAxis : BOOL; //Es werden alle Tools an der selben Achse betrachtet, ansonsten werden nur das Tool selber und seine Childs betrachtet	
END_VAR

VAR
	pTempTool : POINTER TO FB_MzTool;
	pTempTool2 : POINTER TO FB_MzTool;
	iter : FB_ObjCollectIteratorDeep;
	stAbsPosTemp : ST_3DPoint;
	stAbsPosTemp2 : ST_3DPoint;
END_VAR
IF bAllOnAxis THEN
	pTempTool := P_pUpperParentTool;
ELSE
	pTempTool := THIS;
END_IF
stAbsPosTemp := pTempTool^.P_stAbsPosPhys;
pTempTool^.P_pObjCollectNode^.nodes.M_GetIterator(iter);
WHILE iter.pNode > 0 DO
	IF iter.pNode^.P_pObject > 0 AND_THEN iter.pNode^.P_pObject^.M_bIsGroup(E_ObjectGroup.OBJECTGROUP_MzTool) THEN
		pTempTool2 := iter.pNode^.P_pObject;
		//Falls das Tool ein ZSensor ist, wird es nur beachtet wenn er auch angebaut ist.
		IF pTempTool2^.P_eObjectType <> E_ObjectType.OBJECTTYPE_ZSensor OR pTempTool2^.P_bSensorMounted THEN
			stAbsPosTemp2 := pTempTool2^.P_stAbsPosPhys;
			IF stAbsPosTemp2.Z < stAbsPosTemp.Z THEN
				stAbsPosTemp := stAbsPosTemp2;
				pTempTool := pTempTool2;
			END_IF			
		END_IF
	END_IF
	iter.M_Increment();
END_WHILE
M_GetClosestTool := pTempTool;
END_METHOD

METHOD M_GetMaxSpeed : REAL
VAR_INPUT
	eDirection : E_MoveDirection;
END_VAR
IF eDirection = E_MoveDirection.DIRECTION_ZMINUS OR eDirection = E_MoveDirection.DIRECTION_ZPLUS THEN
	IF pZAxisRef > 0 THEN
		M_GetMaxSpeed := pZAxisRef^.P_rMaxSpeed;
	END_IF
ELSE
	M_GetMaxSpeed := SUPER^.M_GetMaxSpeed(eDirection);
END_IF
END_METHOD

METHOD M_GetMinMaxActPos
VAR_INPUT
	pData : POINTER TO ARRAY[0..19] OF DINT;
END_VAR
VAR
	stCurrPosTotal : ST_3DPoint;
END_VAR
SUPER^.M_GetMinMaxActPos(pData);

//Z weiter verrechnen
pData^[4] := pData^[4] + REAL_TO_DINT(pZAxisRef^.P_rMinPos);
pData^[5] := pData^[5] + REAL_TO_DINT(pZAxisRef^.P_rMaxPos);
stCurrPosTotal := P_stCurrentPosTotal;
pData^[6] := REAL_TO_DINT(stCurrPosTotal.X);
pData^[7] := REAL_TO_DINT(stCurrPosTotal.Y);
pData^[8] := REAL_TO_DINT(stCurrPosTotal.Z);
END_METHOD

METHOD M_GetNozzle : POINTER TO FB_Nozzle
VAR_INPUT
END_VAR

VAR
	the: INT;
END_VAR
IF pPiece > 0 THEN
	IF pPiece^.P_eObjectType = E_ObjectType.OBJECTTYPE_Nozzle THEN
		M_GetNozzle := pPiece;
	END_IF
END_IF
END_METHOD

METHOD M_GetZAxisRef : POINTER TO FB_ZAxisRef
VAR_INPUT
	pTool : POINTER TO FB_MzTool;
	pToolSlot : POINTER TO FB_Slot;
END_VAR
M_GetZAxisRef := pParentMzTool^.M_GetZAxisRef(pTool, pParentSlot);
END_METHOD

METHOD M_RawPosToRealPos : ST_3DPoint
VAR_INPUT
	stRawPos : ST_3DPoint;
END_VAR

VAR
	stTemp		: ST_3DPoint;
	stAbsPos : ST_3DPoint;
END_VAR
stAbsPos := P_stAbsPosTotal;
stTemp.X := stRawPos.X + stAbsPos.X;
stTemp.Y := stRawPos.Y + stAbsPos.Y;
stTemp.Z := stAbsPos.Z - stRawPos.Z;
M_RawPosToRealPos := stTemp;
END_METHOD

METHOD M_RemoveChild : ERRORID
VAR_INPUT
	pObject	: POINTER TO FB_Object;
END_VAR

VAR
END_VAR
M_RemoveChild := SUPER^.M_RemoveChild(pObject);
IF M_RemoveChild = 0 AND pObject^.M_bIsGroup(E_ObjectGroup.OBJECTGROUP_Piece) THEN
	pPiece := 0;
END_IF
END_METHOD

METHOD M_SetAllProps : ERRORID
VAR_INPUT
	refCmdData : REFERENCE TO  ST_CmdData;
END_VAR
M_SetAllProps := SUPER^.M_SetAllProps(refCmdData);
IF M_SetAllProps > 0 THEN
	RETURN;
END_IF

//ZAxisRef vom Parent holen
pZAxisRef := pParentMzTool^.M_GetZAxisRef(THIS, pParentSlot);

IF pZAxisRef = 0 THEN
	M_SetAllProps := E_ErrorIdObjMgmt.ERRORID_InvalidAxisRef;
	RETURN;
END_IF

pZAxisRef^.bHasTool := TRUE;

pXDrive := pParentMzTool^.P_pXDrive;
pYDrive := pParentMzTool^.P_pYDrive;
pFbMultiZ := pParentMzTool^.P_pFbMultiZ;
END_METHOD

METHOD M_SetCurrentPos
VAR_INPUT
	nDimension : USINT;
	rValue : REAL;
END_VAR

VAR
	rAbsPos : REAL;
	stAbsPosParent : ST_3DPoint;
	stHelpPoint : ST_3DPoint;
END_VAR
IF nDimension = 1 THEN //X
	rAbsPos := rValue - pXDrive^.P_rActPos;
	stOffset.X := 0;
	IF pParentMzTool > 0 THEN
		stAbsPosParent := pParentMzTool^.P_stAbsPosTotal;
	END_IF
	stRelPos.X := rAbsPos - stAbsPosParent.X;
ELSIF nDimension = 2 THEN //Y
	rAbsPos := rValue - pYDrive^.P_rActPos;
	stOffset.Y := 0;
	IF pParentMzTool > 0 THEN
		stAbsPosParent := pParentMzTool^.P_stAbsPosTotal;
	END_IF
	stRelPos.Y := rAbsPos - stAbsPosParent.Y;
ELSIF nDimension = 3 THEN //Z
	stOffset.Z := 0;
	stHelpPoint := P_stAbsPosTotal;
	IF eObjectType <> E_ObjectType.OBJECTTYPE_MZHead THEN
		IF pParentMzTool > 0 THEN
			stAbsPosParent := pParentMzTool^.P_stAbsPosTotal;
		END_IF
		rAbsPos := pZAxisRef^.P_rCurrentPos + rValue;
	END_IF
	stRelPos.Z := rAbsPos - stAbsPosParent.Z;
END_IF
END_METHOD

METHOD M_UpdateParent
VAR_INPUT
END_VAR

VAR
	pObject : POINTER TO FB_Object;
END_VAR
IF pObjCollectNode > 0 AND_THEN pObjCollectNode^.pOwnerColl > 0 THEN
	pObject := pObjCollectNode^.P_pOwnerColl^.pOwnerNode^.P_pObject;	
END_IF

IF pObject > 0 THEN
	pParentMzTool := pObject;
	pParentSlot := pObject^.M_GetSlotFromChild(THIS);
ELSE
	pParentMzTool := 0;
	pParentSlot := 0;
END_IF
END_METHOD

PROPERTY P_bCollFree : BOOL
GET
VAR
	st3DPoint 		: ST_3DPoint;
	rAbsZOffsetHead	: REAL;
END_VAR
//Ermittlung, ob Tool in kollisionsfreiem Bereich
//Kollisionsfreihheit ist gegeben, wenn Unterkante Z-Wert von Tool >= kollissiongefährdete Höhe Workplate
//MzHead und die Tools unterhalb der Workplate sind immer kollisionsfrei
IF eObjectType = E_ObjectType.OBJECTTYPE_MZHead THEN
	P_bCollFree := TRUE;
ELSE
	IF NOT P_pMzHead^.P_bIsTopHead THEN
		P_bCollFree := TRUE;
		RETURN;
	END_IF
	
	IF NOT bInitAxisOk THEN
		P_bCollFree := FALSE;
		RETURN;
	END_IF
	
	//Aktuelle Position Tool ermitteln
	st3DPoint := P_stCurrentPosPhys;
	st3DPoint.Z := st3DPoint.Z + 11;
	IF st3DPoint.Z >  pAssignWorkplate^.P_rCollHeight THEN
		P_bCollFree := TRUE;
	END_IF
	
END_IF
END_GET
END_PROPERTY

PROPERTY P_bIsInit : BOOL
GET
P_bIsInit := bInitAxisOk AND pZAxisRef^.stStatus.bIsHomed;
END_GET
END_PROPERTY

PROPERTY P_bIsMESTool : BOOL
GET
P_bIsMESTool := bIsMESTool;
END_GET
END_PROPERTY

PROPERTY P_bSensorMounted : BOOL
GET
END_GET
END_PROPERTY

PROPERTY P_bXYIsMoving : BOOL
GET
VAR
	i		: UINT;
	bTemp	: BOOL;
END_VAR
P_bXYIsMoving:= bXYIsMoving;
END_GET
SET
bXYIsMoving := P_bXYIsMoving;
END_SET
END_PROPERTY

PROPERTY P_nParentObjectId : UINT
GET
IF pParentMzTool > 0 THEN
	P_nParentObjectId := pParentMzTool^.P_nObjectID;
END_IF
END_GET
END_PROPERTY

PROPERTY P_nReducedMoveZDist : DINT
GET
P_nReducedMoveZDist := nReducedMoveZDist;
END_GET
SET
nReducedMoveZDist := P_nReducedMoveZDist;
END_SET
END_PROPERTY

PROPERTY P_nReducedMoveZSpeed : DINT
GET
P_nReducedMoveZSpeed := nReducedMoveZSpeed;
END_GET
SET
nReducedMoveZSpeed := P_nReducedMoveZSpeed;
END_SET
END_PROPERTY

PROPERTY P_nZAxisNr : USINT
GET
IF pZAxisRef > 0 THEN
	P_nZAxisNr := pZAxisRef^.nChannel;
END_IF
END_GET
END_PROPERTY

PROPERTY P_pMzHead : POINTER TO FB_MzHead
GET
P_pMzHead := pParentMzTool^.P_pMzHead;
END_GET
END_PROPERTY

PROPERTY P_pParentMzTool : POINTER TO FB_MzBase
GET
P_pParentMzTool := pParentMzTool;
END_GET
END_PROPERTY

//Das Tool, was als Parent den Head hat bzw. direkt an der Achse befindet
PROPERTY P_pUpperParentTool : POINTER TO FB_MzTool
GET
VAR
	pTool : POINTER TO FB_MzTool;
END_VAR
IF pParentMzTool^.P_eObjectType = E_ObjectType.OBJECTTYPE_MZHead THEN
	P_pUpperParentTool := THIS;
ELSE
	pTool := pParentMzTool;
	P_pUpperParentTool := pTool^.P_pUpperParentTool;
END_IF
END_GET
END_PROPERTY

PROPERTY P_pZAxisRef : POINTER TO FB_ZAxisRef
GET
P_pZAxisRef := pZAxisRef;
END_GET
END_PROPERTY

PROPERTY P_rToolRadius : REAL
GET
VAR
	stDim : ST_3DDimension;
END_VAR
//Manche abgeleitete Tools definieren ihren eigenen Tool-Radius
IF pPiece > 0 THEN
	stDim := pPiece^.P_stDimension;
	P_rToolRadius := stDim.Width / 2.0;
ELSE
	P_rToolRadius := 10000.0;	
END_IF
END_GET
END_PROPERTY

PROPERTY P_stAbsPosPhys : ST_3DPoint
GET
VAR
	stTemp	: ST_3DPoint;
	stDim	: ST_3DDimension;
END_VAR
//Die absolute Postion eines Tool in "Z" hat nicht den gleichen Bezug wie X und Y
//X und Y beziehen sich auf den Koordinatenursprung, wenn die Achsen theoretisch aus Antrieb (0;0) stehen
//Z bezieht sich auf die Sliderunterkante des Z-Antriebes verechnet mit AbsPos vom Head(Ergebnis ist in den meisten Fällen negativ)

stTemp := F_Add3DPoints(stRelPos,stOffset);
//Offsets der Pieces verrechnen
IF pPiece > 0 THEN
	stDim := pPiece^.P_stDimension;
	IF NOT pPiece^.P_bIgnoreOffset THEN
		stTemp := F_Add3DPoints(stTemp,pPiece^.P_stOffset);	
	END_IF
	stTemp.Z := stTemp.Z + pPiece^.P_rZOverlapTool - stDim.Height;
	IF pPiece^.P_pParentSlot > 0 THEN
		stTemp := F_Add3DPoints(stTemp,pPiece^.P_pParentSlot^.P_stRelPos);
	END_IF
END_IF
//AbsPos vom ParentSlot holen
IF pParentSlot > 0 THEN
	stTemp := F_Add3DPoints(stTemp,pParentSlot^.P_stAbsPos);
END_IF

P_stAbsPosPhys := stTemp;
END_GET
END_PROPERTY

PROPERTY P_stAbsPosPhysExclPiece : ST_3DPoint
GET
VAR
	stTemp	: ST_3DPoint;
END_VAR
//Die absolute Postion eines Tool in "Z" hat nicht den gleichen Bezug wie X und Y
//X und Y beziehen sich auf den Koordinatenursprung, wenn die Achsen theoretisch aus Antrieb (0;0) stehen
//Z bezieht sich auf die Sliderunterkante des Z-Antriebes verechnet mit AbsPos vom Head(Ergebnis ist in den meisten Fällen negativ)

stTemp := F_Add3DPoints(stRelPos,stOffset);
//AbsPos vom ParentSlot holen
IF pParentSlot > 0 THEN
	stTemp := F_Add3DPoints(stTemp,pParentSlot^.P_stAbsPos);
END_IF

P_stAbsPosPhysExclPiece := stTemp;
END_GET
END_PROPERTY

PROPERTY P_stCurrentPosPhys : ST_3DPoint
GET
VAR
	stTemp		: ST_3DPoint;
	stAbsPos : ST_3DPoint;
END_VAR
stAbsPos := P_stAbsPosPhys;
stTemp.X := pXDrive^.P_rActPos + stAbsPos.X;
stTemp.Y := pYDrive^.P_rActPos + stAbsPos.Y;

IF pZAxisRef > 0  THEN
	stTemp.Z := stAbsPos.Z + pZAxisRef^.P_rCurrentPos;
END_IF
P_stCurrentPosPhys := stTemp;
END_GET
END_PROPERTY

PROPERTY P_stCurrentXYArea : FB_RectAngle
GET
VAR
	stPoint : ST_3DPoint;
END_VAR
stPoint := P_stCurrentPosPhys;
P_stCurrentXYArea.X1 := stPoint.X - 1.0;
P_stCurrentXYArea.X2 := stPoint.X + 1.0;
P_stCurrentXYArea.Y1 := stPoint.Y - 1.0;
P_stCurrentXYArea.Y2 := stPoint.Y + 1.0;
END_GET
END_PROPERTY

END_FUNCTION_BLOCK

// ---- Objects/Tools/FB_MzBase.TcPOU
FUNCTION_BLOCK FB_MzBase EXTENDS FB_Object IMPLEMENTS I_Device

VAR_OUTPUT
	bBusy				: BOOL;
END_VAR

VAR
	bInitFB				: BOOL := TRUE;			//zum erstmaligen Initialisieren des FB
	

	fbSlotList			: FB_SlotList;
	nNumberOfSlots		: UINT;
	nFirstSlotPropIndex	: UINT;	//erster Index für Slots (benötigt in M_SetSingleProps)
	nLastSlotPropIndex	: UINT;	//letzte Index für Slots (benötigt in M_SetSingleProps)
	
	//Variablen allgemeine Statemachine
	bCanceled			: BOOL;
	bError				: BOOL;
	stError				: ST_Error;
	bStopAllOnError		: BOOL;
	eCurrentState		: E_MachineState := E_MachineState.MACHINESTATE_Idle;
	i					: UINT;					//allg. Zählvariable

	nDeviceIdx			: UINT;			//eigener Index in aI_Device[Idx]
	nCurrentPropIndex	: UINT;

	nSpecPropIndex		: UINT;			//erster Index für Specialproperties (ab direkter Erbe von FB_MzTool) (benötigt in M_SetSingleProps + M_GetSingleProp)
	
	pAssignWorkplate	: POINTER TO FB_Workplate;
	nNotifyId			: UINT;
	stRelPos			: ST_3DPoint;	//Relative Position zum Parent
	stOffset			: ST_3DPoint;	//Offset

	
	pFbMultiZ			: POINTER TO FB_MultiZRef;
	pXDrive				: POINTER TO FB_XYDriveBase;
	pYDrive				: POINTER TO FB_XYDriveBase;
	pPiece				: POINTER TO FB_PieceBase;

	//****************************************Aktionvariablen****************************************************
	
	//Verkettete Liste für BasicActions
	fbList				: FB_LinkedListCtrl;
	hList				: T_HLINKEDLIST;
	aNodes           	: ARRAY[0..4] OF T_LinkedListEntry;
	getValue			: PVOID;
	getPosPtr       	: POINTER TO T_LinkedListEntry := 0;

	//Action: "InitBase"
	bInitAxisOk			: BOOL;
	bInitToolOk			: BOOL;
	bInitAxis			: BOOL;
	bReInit				: BOOL;
	nStateA_InitAxis	: USINT;			//State von A_Init() BasisFb
	bInitReadyX			: BOOL;
	bInitReadyY			: BOOL;
	bInitErrorX			: BOOL;
	bInitErrorY			: BOOL;
	fbZmHome			: FB_ZM_Home;
	nCurInitZAxis		: USINT;
	timeoutInit			: TON;
	
	bMeasured			: BOOL;				//als Merker, ob bei Tipvermessung bereits komplette Vermessung durchgeführt wurde
	bDisableFreeMove	: BOOL;
	
	//Action: "JogXY"
	bJogXY				: BOOL;
	nStateA_JogXY		: USINT;			//State von A_JogXY()
	eJogXYDirectionNew	: E_MoveDirection;
	eJogXYDirection		: E_MoveDirection;
	nCurrentJogXYAxis	: USINT;			//1= X, 2=Y, 3=Z;(Z wird in FB_MzTool verarbeitet)
	bJogXYForward		: BOOL;
	bJogXYBackwards		: BOOL;
	bJogXYClock			: BOOL;
	bJogXYModeInchingNew: BOOL;				//wenn True dann Tipbetrieb sonst kontinuierlich
	bJogXYModeInching	: BOOL;				//wenn True dann Tipbetrieb sonst kontinuierlich
	rJogXYDistance		: REAL;
	rJogXYSpeed			: REAL;
	bJogXYImpuls		: BOOL;	
	
	//Action: "MoveX"
	bMoveX				: BOOL;
	nStateA_MoveX		: USINT;			//State von A_MoveX()
	bFlagMoveX			: BOOL := TRUE;		//Hilfsflag
	
	//Action: "MoveY"	
	bMoveY				: BOOL;
	nStateA_MoveY		: USINT;			//State von A_MoveX()
	bFlagMoveY			: BOOL := TRUE;		//Hilfsflag
	
	//Action: "MoveXY"	
	bMoveXY				: BOOL;
	nStateA_MoveXY		: USINT;			//State von A_MoveXY()
	bFlagMoveXY			: BOOL := TRUE;		//Hilfsflag
	bMoveXReady			: BOOL;
	bMoveXError			: BOOL;
	bMoveYReady			: BOOL;
	bMoveYError			: BOOL;
	bMoveXYReady		: BOOL;
	recteMoveRange		: FB_Rectangle;
	pHighestTarget		: POINTER TO FB_TargetBase;
	bSynchron			: BOOL;	//beide Achsen kommen zeitgleich an
	stCurrentPosPhys	: ST_3DPoint;
	
	//Action: "MoveZ"
	bMoveZ				: BOOL;
	nStateA_MoveZ		: USINT;			//State von A_Move()
	bFlagMoveZ			: BOOL := TRUE;		//Hilfsflag
	eMoveModeZ			: E_MoveMode;
	
	fbZmMove			: FB_ZM_Move;
	fbZmStop			: FB_ZM_Stop;

	//Action: "Move allgemein"
	eMoveMode			: E_MoveMode;
	bMoveModeXYRelativ	: BOOL;
	rMovePositionX		: REAL;
	rMovePositionY		: REAL;
	rMovePositionZ		: REAL;
	rMoveSpeedX			: REAL;
	rMoveSpeedY			: REAL;
	rMoveSpeedZ			: REAL;
	rDistanceX			: REAL;
	rDistanceY			: REAL;
	st3DPoint			: ST_3DPoint;
	st3DPoint1			: ST_3DPoint;
	//stDimension			: ST_3DDimension;
	stAreaCollFree		: FB_Rectangle;		//kollisionsfreier XY-Bereich um die aktuelle XY-Position des Tools(wird bei Z-Zustellung gesetzt)
	bIgnoreZCollision	: BOOL;
	eCrashAvoidanceMode	: E_CrashAvoidanceMode;
	stActionData		: ST_ActionData;
	bZIsMoving			: BOOL;
	bXYIsMoving			: BOOL;
	pMtp				: POINTER TO FB_Mtp;
	pHead				: POINTER TO FB_MzHead;
	pCustomUnitType1	: POINTER TO FB_CustomUnitType1;
	
	//Action: "Stop"
	bStop				: BOOL;
	nStateA_Stop		: USINT;			//State von A_Stop()
	bFlagStop			: BOOL := TRUE;		//Hilfsflag
	
	//Action: "Reset"
	nStateA_ResetBase	: USINT;			//State von A_Reset() BasisFB
	nStateA_ResetTool	: USINT;
	nStateA_ResetSpec	: USINT;			//State von A_Reset() SpecialFB
	bFlagA_ResetBase	: BOOL := TRUE;		//Hilfsflag von A_Reset() BasisFB
	bFlagA_ResetSpec	: BOOL := TRUE;		//Hilfsflag von A_Reset() SpecialFB
	timeoutReset		: TON;
	
	//Prozessdaten
	stProcessData		: ST_ObjectProcData;	//werden am Ende in globales Array übertragen, welches per Notifiction zum PC übertragen werden 
	stCurrentPos		: ST_3DPoint;
	
END_VAR

IF bInitFB THEN
	bInitFB := FALSE;
	F_CreateLinkedListHnd( ADR( aNodes ), SIZEOF( aNodes ), hList );
	stError.ObjectId := nObjectID;
	stError.HardwareGrp := E_HardwareGrp.Nothing;
END_IF

CASE eCurrentState OF
	E_MachineState.MACHINESTATE_Active:
		bBusy := TRUE;
		IF bInitAxis THEN	//Initialisieren
			A_Init();
			IF nStateA_InitAxis >= 80 THEN
				IF nStateA_InitAxis >= 99 THEN
					bError := TRUE;
				END_IF
				bInitAxis := FALSE;
				nStateA_InitAxis := 0;
				M_RemoveListEntry(nSearchValue:= E_Action.ACTION_Init);
			END_IF
		END_IF
		
		IF bJogXY THEN	//Joggen
			A_JogXY();
			IF nStateA_JogXY >= 80 THEN
				IF nStateA_JogXY >= 99 THEN
					bError := TRUE;
				END_IF
				bJogXY := FALSE;
				nStateA_JogXY := 0;
				M_RemoveListEntry(nSearchValue:= E_Action.ACTION_Jog);
			END_IF
		END_IF

		IF bMoveX THEN	//Move X absolut oder relativ
			A_MoveX();
			IF nStateA_MoveX >= 80 THEN
				IF nStateA_MoveX >= 99 THEN
					bStopAllOnError := TRUE; 
					bError := TRUE;
				END_IF
				bMoveX := FALSE;
				bXYIsMoving := FALSE;
				nStateA_MoveX := 0;
				M_RemoveListEntry(nSearchValue:= E_Action.ACTION_MoveX);
			END_IF
		END_IF		
		
		IF bMoveY THEN	//Move Y absolut oder relativ
			A_MoveY();
			IF nStateA_MoveY >= 80 THEN
				IF nStateA_MoveY >= 99 THEN
					bStopAllOnError := TRUE;
					bError := TRUE;
				END_IF
				bMoveY := FALSE;
				bXYIsMoving := FALSE;
				nStateA_MoveY := 0;
				M_RemoveListEntry(nSearchValue:= E_Action.ACTION_MoveY);
			END_IF
		END_IF	

		IF bMoveXY THEN	//Move XY absolut oder relativ
			A_MoveXY();
			IF nStateA_MoveXY >= 80 THEN
				IF nStateA_MoveXY >= 99 THEN
					bStopAllOnError := TRUE; 
					bError := TRUE;
				END_IF
				bMoveXY := FALSE;
				bXYIsMoving := FALSE;
				nStateA_MoveXY := 0;
				M_RemoveListEntry(nSearchValue:= E_Action.ACTION_MoveXY);
			END_IF
		END_IF
		
		IF bMoveZ THEN	//Move Z absolut oder relativ
			A_MoveZ();
			IF nStateA_MoveZ >= 80 THEN
				IF nStateA_MoveZ >= 99 THEN
					bStopAllOnError := TRUE;
					bError := TRUE;
				END_IF
				bMoveZ := FALSE;
				bZIsMoving := FALSE;
				nStateA_MoveZ := 0;
				M_RemoveListEntry(nSearchValue:= E_Action.ACTION_MoveZ);
			END_IF
		END_IF		
		
		IF bStop THEN	//alle Actions stoppen
			A_Stop();
			IF nStateA_Stop >= 80 THEN
				IF nStateA_Stop >= 99 THEN
					bError := TRUE;					
				END_IF
				M_RemoveListEntry(nSearchValue:= E_Action.ACTION_Stop);
				bStop := FALSE;
				nStateA_Stop := 0;
				bCanceled := TRUE;
			END_IF							
		END_IF

		IF hList.nCount = 0 THEN
			eCurrentState := E_MachineState.MACHINESTATE_Ready;
		END_IF
		
		IF bError THEN
			IF hList.nCount > 1 THEN	//mehr Aktionen als die den Fehler verursachende
				bStop := TRUE;
			ELSE
				eCurrentState := E_MachineState.MACHINESTATE_Error;	
			END_IF
		END_IF

	E_MachineState.MACHINESTATE_Reset:
		A_Reset();
		//Wenn A_Reset() in SpezialFB existiert, dann wird sie dort aufgerufen
		//in diesem Fall wird FB_MzBase.A_Reset() von SpezialFB über SUPER^.A_Reset() aufgerufen
		
		IF nStateA_ResetBase >= 80 THEN
			IF nStateA_ResetBase >= 99 THEN
				bError := TRUE;
				eCurrentState := E_MachineState.MACHINESTATE_Error;
			ELSE
				fbList.A_Reset(hList := hList);
				bStopAllOnError := FALSE;
				bError := FALSE;
				eCurrentState := E_MachineState.MACHINESTATE_Idle;
			END_IF
			bBusy := FALSE;
			nStateA_ResetBase := 0;
			nStateA_ResetTool := 0;
			nStateA_ResetSpec := 0;
		END_IF
END_CASE

//Nicht im CASE-Block, damit busy in gleichem Zyklus zurückgesetzt wird		
IF eCurrentState = E_MachineState.MACHINESTATE_Ready THEN
		bBusy := FALSE;
		eCurrentState := E_MachineState.MACHINESTATE_Idle;
ELSIF eCurrentState = E_MachineState.MACHINESTATE_Error THEN
		bBusy := FALSE;
END_IF

//Prozessdaten aktualisieren
stProcessData.nObjId := nObjectID;
stProcessData.n32Data[0] := BOOL_TO_DINT(P_bIsInit);
stProcessData.n32Data[1] := eCurrentState;
stProcessData.n32Data[2] := stError.ErrorId;

ACTION A_Init:
//Initilaisierung erfolgt jeweils in FB_MzTool.A_Init() und FB_XXXX.A_Init()
END_ACTION

ACTION A_JogXY:
IF nStateA_JogXY = 0 THEN
	IF bJogXYModeInching THEN
		nStateA_JogXY := 1;	//Incr
	ELSE
		nStateA_JogXY := 3;	//Continous
	END_IF
END_IF
 
IF nStateA_JogXY = 1 THEN	//incrementellen Jog-Befehl 1x absetzen
	CASE eJogXYDirection OF
		E_MoveDirection.DIRECTION_XPLUS:
			nCurrentJogXYAxis := 1;
			pXDrive^.M_Jog(bForward:= TRUE, bBackward:= FALSE, bInching:= TRUE, rDistance:= rJogXYDistance, rSpeed:= rJogXYSpeed);
			bXYIsMoving := TRUE;
		E_MoveDirection.DIRECTION_XMINUS:	
			nCurrentJogXYAxis := 1;
			pXDrive^.M_Jog(bForward:= FALSE, bBackward:= TRUE, bInching:= TRUE, rDistance:= rJogXYDistance, rSpeed:= rJogXYSpeed);
			bXYIsMoving := TRUE;
			bXYIsMoving := TRUE;
		E_MoveDirection.DIRECTION_YPLUS:
			nCurrentJogXYAxis := 2;
			pYDrive^.M_Jog(bForward:= TRUE, bBackward:= FALSE, bInching:= TRUE, rDistance:= rJogXYDistance, rSpeed:= rJogXYSpeed);
			bXYIsMoving := TRUE;
		E_MoveDirection.DIRECTION_YMINUS:
			nCurrentJogXYAxis := 2;
			pYDrive^.M_Jog(bForward:= FALSE, bBackward:= TRUE, bInching:= TRUE, rDistance:= rJogXYDistance, rSpeed:= rJogXYSpeed);
			bXYIsMoving := TRUE;
	END_CASE
	nStateA_JogXY := 2;
END_IF

IF nStateA_JogXY = 2 THEN //warten bis inkrementelles Joggen fertig bzw auf neuen Befehl warten
	IF NOT bJogXYModeInching THEN //Wechseln zu kontinulierlichem Joggen
		nStateA_JogXY := 3;
	END_IF
	
	IF eJogXYDirection = E_MoveDirection.DIRECTION_STOP THEN
		nStateA_JogXY := 4;
	END_IF
END_IF

IF nStateA_JogXY = 3 THEN //zyklisches Absetzen des kontinuierlichen Jog-Befehls, hier kann auch Stop abgesetzt werden, bzw neuer inkr. Befehl
	IF bJogXYImpuls THEN
		CASE eJogXYDirection OF
			E_MoveDirection.DIRECTION_STOP:
				nStateA_JogXY := 4;
			E_MoveDirection.DIRECTION_XPLUS:
				nCurrentJogXYAxis := 1;
				pXDrive^.M_Jog(bForward:= TRUE, bBackward:= FALSE, bInching:= FALSE, rDistance:= rJogXYDistance, rSpeed:= rJogXYSpeed);
				bXYIsMoving := TRUE;
			E_MoveDirection.DIRECTION_XMINUS:	
				nCurrentJogXYAxis := 1;
				pXDrive^.M_Jog(bForward:= FALSE, bBackward:= TRUE, bInching:= FALSE, rDistance:= rJogXYDistance, rSpeed:= rJogXYSpeed);
				bXYIsMoving := TRUE;
				bXYIsMoving := TRUE;
			E_MoveDirection.DIRECTION_YPLUS:
				nCurrentJogXYAxis := 2;
				pYDrive^.M_Jog(bForward:= TRUE, bBackward:= FALSE, bInching:= FALSE, rDistance:= rJogXYDistance, rSpeed:= rJogXYSpeed);
				bXYIsMoving := TRUE;
			E_MoveDirection.DIRECTION_YMINUS:
				nCurrentJogXYAxis := 2;
				pYDrive^.M_Jog(bForward:= FALSE, bBackward:= TRUE, bInching:= FALSE, rDistance:= rJogXYDistance, rSpeed:= rJogXYSpeed);
				bXYIsMoving := TRUE;
		END_CASE
	END_IF
	bJogXYImpuls := FALSE;
END_IF

IF nStateA_JogXY = 4 THEN //Stop
	pXDrive^.M_Jog(bForward:= FALSE, bBackward:= FALSE, bInching:= FALSE, rDistance:= 0.0, rSpeed:= 0.0);
	pYDrive^.M_Jog(bForward:= FALSE, bBackward:= FALSE, bInching:= FALSE, rDistance:= 0.0, rSpeed := 0.0);
	//IF bJogXYModeInching THEN
		pXDrive^.M_Stop();
		pYDrive^.M_Stop();
	//END_IF
	nStateA_JogXY := 5;
END_IF

//Abfragen, ob Jogging fertig
IF nCurrentJogXYAxis = 1 THEN	//X
	IF NOT pXDrive^.P_bBusy THEN
		IF pXDrive^.P_bError THEN
			stError.ErrorId := pXDrive^.P_nErrorId;
			stError.HardwareGrp := E_HardwareGrp.AxisX;
			stError.HardwareNr	:= 1;
			stError.POUState := nStateA_JogXY;
			nStateA_JogXY := 99;
		ELSE
			nStateA_JogXY := 80;	
		END_IF
		nCurrentJogXYAxis := 0;
		bXYIsMoving := FALSE;
	END_IF
ELSIF nCurrentJogXYAxis = 2 THEN	//Y
	IF NOT pYDrive^.P_bBusy THEN
		IF pYDrive^.P_bError THEN
			stError.ErrorId := pYDrive^.P_nErrorId;
			stError.HardwareGrp := E_HardwareGrp.AxisY;
			stError.HardwareNr	:= 1;
			stError.POUState := nStateA_JogXY;
			nStateA_JogXY := 99;
		ELSE
			nStateA_JogXY := 80;	
		END_IF
		nCurrentJogXYAxis := 0;
		bXYIsMoving := FALSE;
	END_IF
ELSE
	nStateA_JogXY := 80;
END_IF

//Errorhandling
IF nStateA_JogXY = 99 THEN
	stError.Cmd := E_Action.ACTION_Jog;
	stError.POU := E_POU.POU_FB_MzBase;
	stError.POUAction := E_POUACT.POUACT_A_JogXY;
	fbErrorList.M_Add(stError);
END_IF
END_ACTION

ACTION A_MoveX:
stError.POUState := nStateA_MoveX;

CASE nStateA_MoveX OF
	0:	
		IF NOT bIgnoreZCollision THEN
			//Distanz ermitteln, für ev. Freifahren der Z-Achsen
			IF eMoveMode = E_MoveMode.MODE_Relative THEN
				rDistanceX := rMovePositionX;
			ELSIF eMoveMode = E_MoveMode.MODE_AbsWithOffset THEN
				st3DPoint := P_stCurrentPosTotal;
				rDistanceX := ABS(rMovePositionX - st3DPoint.X);
			ELSIF eMoveMode = E_MoveMode.MODE_AbsNoneOffset THEN
				rDistanceX := ABS(rMovePositionX - pXDrive^.P_rActPos);
			END_IF
			
			stActionData.eAction := E_Action.ACTION_MoveZ;
			stActionData.aParams[1] := E_MoveMode.MODE_Free;
			stActionData.aParams[3] := -1;
			
			//Bei MoveX müssen definitiv die Achsen aller Heads kollisionsfrei sein
			nStateA_MoveX := 1;
			FOR i:= 1 TO fbObjectDirectory.nCntMZHead BY 1 DO
				IF NOT afbMzHead[i].P_bCollFree THEN
					stError.ErrorId := afbMzHead[i].M_ExeAction(stActionData);
					IF stError.ErrorId > 0 THEN
						stError.HardwareGrp := E_HardwareGrp.AxisZ;
						stError.HardwareNr := 0;
						nStateA_MoveX := 99;
						EXIT;
					END_IF
				END_IF
			END_FOR
		ELSE
			nStateA_MoveX := 2;
		END_IF
		
	1:	//warten bis beide Köpfe fertig
		nStateA_MoveX := 2;
		FOR i:= 1 TO fbObjectDirectory.nCntMZHead BY 1 DO
			IF afbMzHead[i].M_GetActionBusy(E_Action.ACTION_MoveZ) THEN
				nStateA_MoveX := 1;
			END_IF
			IF afbMzHead[i].P_bError THEN
				stError.ErrorId := afbMzHead[i].P_nErrorId;
				stError.HardwareGrp := E_HardwareGrp.AxisZ;
				nStateA_MoveX := 99;
				EXIT;
			END_IF
		END_FOR			
		
	2:	//In Abhängigkeit von MoveMode absolut oder relativ fahren
		IF eMoveMode = E_MoveMode.MODE_Relative THEN	//Relativ
			stError.ErrorId := pXDrive^.M_MoveRel(rDistance:= rMovePositionX, rSpeed:= rMoveSpeedX, rAcceleration:= 0.0, rDeceleration:= 0.0);
			nStateA_MoveX := 3; 
		ELSIF eMoveMode = E_MoveMode.MODE_AbsWithOffset THEN	//Absolut mit Offsets
			//Achsenposition berechnen
			//Position ergibt sich aus Zielposition abzüglich aller Offsets
			st3DPoint := P_stAbsPosTotal;	//Summe aller Offsets
			rMovePositionX := rMovePositionX - st3DPoint.X;
			stError.ErrorId := pXDrive^.M_MoveAbs(rPosition:= rMovePositionX, rSpeed:= rMoveSpeedX, rAcceleration:= 0.0, rDeceleration:= 0.0);
			nStateA_MoveX := 3; 
		ELSIF eMoveMode = E_MoveMode.MODE_AbsNoneOffset THEN	//Absolut OHNE Offsets!!
			stError.ErrorId := pXDrive^.M_MoveAbs(rPosition:= rMovePositionX, rSpeed:= rMoveSpeedX, rAcceleration:= 0.0, rDeceleration:= 0.0);
 			nStateA_MoveX := 3;
		ELSIF eMoveMode = E_MoveMode.MODE_Home THEN	//auf 0 fahren
			stError.ErrorId := pXDrive^.M_MoveAbs(rPosition:= 0.0, rSpeed:= rMoveSpeedX, rAcceleration:= 0.0, rDeceleration:= 0.0);
 			nStateA_MoveX := 3;
		ELSE
			nStateA_MoveX := 99; //Error (Dieser Fall sollte nicht auftreten. MoveMode wird in M_ExeAction() abgefangen)
		END_IF
		
		IF stError.ErrorId > 0 THEN
			stError.HardwareGrp := E_HardwareGrp.AxisX;
			nStateA_MoveX := 99;
		END_IF
		
	3:	//Warten bis Positionierung fertig
		IF NOT pXDrive^.P_bBusy THEN
			IF pXDrive^.P_bError THEN
				stError.ErrorId := pXDrive^.P_nErrorId;
				stError.HardwareNr	:= 1;
				//fbXDrive resetten!!
 				nStateA_MoveX := 99;
			ELSE
				nStateA_MoveX := 80;
			END_IF
		END_IF
	
	70:	//Stoppen
		pXDrive^.M_Stop();
		IF NOT pXDrive^.P_bBusy THEN
			nStateA_MoveX := 80;
		END_IF
END_CASE

//Errorhandling
IF nStateA_MoveX = 99 THEN
	stError.ObjectId := nObjectID;
	stError.Cmd := E_Action.ACTION_MoveX;
	stError.POU := E_POU.POU_FB_MzBase;
	stError.POUAction := E_POUACT.POUACT_A_MoveX;
	fbErrorList.M_Add(stError);
END_IF
END_ACTION

ACTION A_MoveXY:
stError.POUState := nStateA_MoveXY;

//States sind in separaten IF-Blöcken, um Zyklen zu sparen
IF nStateA_MoveXY = 0 THEN
	stCurrentPosPhys := P_stCurrentPosPhys;
	nStateA_MoveXY := 1;
	//Distanz ermitteln, für ev. Freifahren der Z-Achsen
	IF eMoveMode = E_MoveMode.MODE_Relative THEN
		rDistanceX := rMovePositionX;
		rDistanceY := rMovePositionY;
	ELSIF eMoveMode = E_MoveMode.MODE_AbsWithOffset THEN
		st3DPoint := P_stCurrentPosTotal;
		rDistanceX := ABS(rMovePositionX - st3DPoint.X);
		rDistanceY := ABS(rMovePositionY - st3DPoint.Y);
	ELSIF eMoveMode = E_MoveMode.MODE_AbsNoneOffset THEN
		rDistanceX := ABS(rMovePositionX - pXDrive^.P_rActPos);
		rDistanceY := ABS(rMovePositionY - pYDrive^.P_rActPos);
	END_IF
	
	IF eCrashAvoidanceMode = E_CrashAvoidanceMode.MoveAllFree THEN
		stActionData.eAction := E_Action.ACTION_MoveZ;
		stActionData.aParams[1] := E_MoveMode.MODE_Free;
		stActionData.aParams[3] := -1; //MaxSpeed
		
		//Die Achsen ermitteln, bei denen der CollFreeArea in den Verfahrweg passt
		//und diese dann vom Freifahren ausschließen
		
		//Wenn nur X-Speed = 0 -> X wird nicht bewegt, dann müssen nur die Achsen des eigenen Heads
		//freigefahren werden
		IF rMoveSpeedX = 0 THEN
			IF NOT P_pMzHead^.M_GetCollFree(rDistanceX,rDistanceY) THEN
				stError.ErrorId := P_pMzHead^.M_ExeAction(stActionData);
				IF stError.ErrorId > 0 THEN
					stError.HardwareGrp := E_HardwareGrp.AxisZ;
					stError.HardwareNr := 0;
					nStateA_MoveXY := 99;
				END_IF
			END_IF
		ELSE
			FOR i:= 1 TO fbObjectDirectory.nCntMZHead BY 1 DO
				IF NOT afbMzHead[i].M_GetCollFree(rDistanceX,rDistanceY) THEN
					stError.ErrorId := afbMzHead[i].M_ExeAction(stActionData);
					IF stError.ErrorId > 0 THEN
						stError.HardwareGrp := E_HardwareGrp.AxisZ;
						stError.HardwareNr := 0;
						nStateA_MoveXY := 99;
					END_IF
				END_IF
			END_FOR				
		END_IF
	ELSIF eCrashAvoidanceMode = E_CrashAvoidanceMode.MoveNoneFree THEN //Crash-Vermeidung ist deaktiviert
		nStateA_MoveXY := 2;
	ELSIF eCrashAvoidanceMode = E_CrashAvoidanceMode.MoveUnusedFree THEN //Alle anderen Tools werden auf FreeHeight gefahren, für sich selbst erfolgt Targetüberwachung
		//Rechteck bilden aus aktueller Position und Zielposition
		//In diesem Rechteck darf sich auf aktueller Höhe kein Target befinden
		recteMoveRange.M_Clear();
		stCurrentPos := P_stCurrentPosTotal;
		 
		IF (rDistanceX > 0.0) THEN
			recteMoveRange.X1 := stCurrentPos.X;
			recteMoveRange.X2 := stCurrentPos.X + rDistanceX + P_rToolRadius;
		ELSE
			recteMoveRange.X2 := stCurrentPos.X;
			recteMoveRange.X1 := stCurrentPos.X + rDistanceX - P_rToolRadius;
		END_IF
		
		IF (rDistanceY > 0.0) THEN
			recteMoveRange.Y1 := stCurrentPos.Y;
			recteMoveRange.Y2 := stCurrentPos.Y + rDistanceY + P_rToolRadius;
		ELSE
			recteMoveRange.Y2 := stCurrentPos.Y;
			recteMoveRange.Y1 := stCurrentPos.Y + rDistanceY - P_rToolRadius;
		END_IF
		
		IF P_pMzHead^.P_bIsTopHead THEN
			pHighestTarget := pAssignWorkplate^.M_GetHighestTarget(recteMoveRange,0.0);	
		END_IF
		
		IF pHighestTarget > 0 THEN //bei unteren Head gibt es kein highest target
			//Ist pHighestTarget eine MTP? und recteMoveRange innerhalb eines Wells?
			IF pHighestTarget^.P_eObjectType = E_ObjectType.OBJECTTYPE_Mtp THEN
				//Mtp erhält einen Methode M_RectIsInnerWell
				pMtp := pHighestTarget;
				IF NOT pMtp^.M_GetRectIsInnerWell(recteMoveRange) THEN
					stError.ErrorId := E_ErrorIdCmd.ERRORID_MoveXYRiskOfCrash;
					nStateA_MoveXY := 99;
				END_IF
			ELSIF pHighestTarget^.P_eObjectType = E_ObjectType.OBJECTTYPE_CustomUnitType1 THEN
				//CustomUnitType1 erhält eine Methode M_RectIsInnerSlot
				pCustomUnitType1 := pHighestTarget;
				IF NOT pCustomUnitType1^.M_GetRectIsInnerSlot(recteMoveRange) THEN
					stError.ErrorId := E_ErrorIdCmd.ERRORID_MoveXYRiskOfCrash;
					nStateA_MoveXY := 99;
				END_IF
			ELSIF pHighestTarget^.P_eObjectType = E_ObjectType.OBJECTTYPE_Slide OR 
					pHighestTarget^.P_eObjectType = E_ObjectType.OBJECTTYPE_SpotArray OR
					pHighestTarget^.P_eObjectType = E_ObjectType.OBJECTTYPE_TargetTray THEN
				IF NOT F_RectInnerRect(recteMoveRange, pHighestTarget^.P_fbAbsRect) THEN
					stError.ErrorId := E_ErrorIdCmd.ERRORID_MoveXYRiskOfCrash;
					nStateA_MoveXY := 99;
				END_IF
			ELSIF pHighestTarget^.P_eObjectType = E_ObjectType.OBJECTTYPE_HighVoltTray THEN
				//Hier sind manchmal Slides in das Tray eingelassen
				IF NOT F_RectInnerRect(recteMoveRange, pHighestTarget^.P_fbAbsRect) THEN
					stError.ErrorId := E_ErrorIdCmd.ERRORID_MoveXYRiskOfCrash;
					nStateA_MoveXY := 99;
				END_IF
			ELSIF (pHighestTarget^.P_rAbsFreeHeight > stCurrentPosPhys.Z) THEN
				stError.ErrorId := E_ErrorIdCmd.ERRORID_MoveXYRiskOfCrash;
				nStateA_MoveXY := 99;
			END_IF
		END_IF
		
		IF nStateA_MoveXY <> 99 THEN
			//Alle anderen Tools freifahren
			IF rMoveSpeedX = 0 THEN	//Falls kein X-Move, dann braucht CoHead nicht freigefahren werden
				IF NOT P_pMzHead^.M_GetCollFree(rDistanceX,rDistanceY) THEN
					stError.ErrorId := P_pMzHead^.M_MoveFree(THIS);
					IF stError.ErrorId > 0 THEN
						stError.HardwareGrp := E_HardwareGrp.AxisZ;
						stError.HardwareNr := 0;
						nStateA_MoveXY := 99;
					END_IF
				END_IF				
			ELSE
				
				IF NOT P_pMzHead^.M_GetCollFree(rDistanceX,rDistanceY) THEN
					stError.ErrorId := P_pMzHead^.M_MoveFree(THIS);
					IF stError.ErrorId > 0 THEN
						stError.HardwareGrp := E_HardwareGrp.AxisZ;
						stError.HardwareNr := 0;
						nStateA_MoveXY := 99;
					END_IF
				END_IF
				
				IF nStateA_MoveXY <> 99 THEN
					IF P_pMzHead^.P_pCoHead > 0 THEN
						IF NOT P_pMzHead^.P_pCoHead^.M_GetCollFree(rDistanceX,rDistanceY) THEN
							stError.ErrorId := P_pMzHead^.P_pCoHead^.M_MoveFree(0);
							IF stError.ErrorId > 0 THEN
								stError.HardwareGrp := E_HardwareGrp.AxisZ;
								stError.HardwareNr := 0;
								nStateA_MoveXY := 99;
							END_IF
						END_IF
					END_IF
				END_IF
			END_IF
		END_IF
	ELSE
		stError.ErrorId := E_ErrorIdCmd.ERRORID_InvalidCrashAvoidanceMode;
		nStateA_MoveXY := 99;
	END_IF
END_IF
		
//warten bis beide Köpfe fertig
IF nStateA_MoveXY = 1 THEN
	//nochmal zu State 0 wechseln, dadurch wird erneut festgestellt, ob alles frei??
	//würde allerdings noch einen Zyklus kosten
	nStateA_MoveXY := 2;
	FOR i:= 1 TO fbObjectDirectory.nCntMZHead BY 1 DO
		IF afbMzHead[i].M_GetActionBusy(E_Action.ACTION_MoveZ) THEN
			nStateA_MoveXY := 1;
		END_IF
		IF afbMzHead[i].P_bError THEN
			stError.ErrorId := afbMzHead[i].P_nErrorId;
			stError.HardwareGrp := E_HardwareGrp.AxisZ;
			nStateA_MoveXY := 99;
			EXIT;
		END_IF
	END_FOR
END_IF

//In Abhängigkeit von MoveMode absolut oder relativ fahren
IF nStateA_MoveXY = 2 THEN
	IF bSynchron THEN
		F_SynchronizeSpeeds(rSpeedSum:= rMoveSpeedX, rDistance1:= rDistanceX, rDistance2:= rDistanceY, rSpeed1:= rMoveSpeedX, rSpeed2 := rMoveSpeedY);	
	END_IF
	nStateA_MoveXY := 3;
	IF eMoveMode = E_MoveMode.MODE_Relative THEN	//Relativ
		stError.ErrorId := pXDrive^.M_MoveRel(rDistance:= rMovePositionX, rSpeed:= rMoveSpeedX, rAcceleration:= 0.0, rDeceleration:= 0.0);
		IF stError.ErrorId > 0 THEN
			stError.HardwareGrp := E_HardwareGrp.AxisX;
			stError.POUState := nStateA_MoveXY;
			nStateA_MoveXY := 99;
		ELSE
			stError.ErrorId := pYDrive^.M_MoveRel(rDistance:= rMovePositionY, rSpeed:= rMoveSpeedY, rAcceleration:= 0.0 ,rDeceleration:= 0.0);
			IF stError.ErrorId > 0 THEN //XDrive muss abgebrochen werden
				pXDrive^.M_Stop();
				stError.HardwareGrp := E_HardwareGrp.AxisY;
				nStateA_MoveXY := 99;
			END_IF
		END_IF
	ELSIF eMoveMode = E_MoveMode.MODE_AbsWithOffset THEN	//Absolut mit Offsets
		//Position ergibt sich aus Zielposition abzüglich aller Offsets
		st3DPoint := P_stAbsPosTotal;	//Summe aller Offsets
		rMovePositionX := rMovePositionX - st3DPoint.X;
		rMovePositionY := rMovePositionY - st3DPoint.Y;
		IF rDistanceX <> 0 THEN
			stError.ErrorId := pXDrive^.M_MoveAbs(rPosition:= rMovePositionX, rSpeed:= rMoveSpeedX ,rAcceleration:= 0.0, rDeceleration:= 0.0);	
		END_IF
		
		IF stError.ErrorId > 0 THEN
			stError.HardwareGrp := E_HardwareGrp.AxisX;
			nStateA_MoveXY := 99;
		ELSE
			IF rDistanceY <> 0 THEN
				stError.ErrorId := pYDrive^.M_MoveAbs(rPosition:= rMovePositionY, rSpeed:= rMoveSpeedY ,rAcceleration:= 0.0, rDeceleration:= 0.0);	
			END_IF
			IF stError.ErrorId > 0 THEN //XDrive muss abgebrochen werden
				pXDrive^.M_Stop();
				stError.HardwareGrp := E_HardwareGrp.AxisY;
				nStateA_MoveXY := 99;
			END_IF
		END_IF
	ELSIF eMoveMode = E_MoveMode.MODE_AbsNoneOffset THEN	//Absolut OHNE Offsets!!
		stError.ErrorId := pXDrive^.M_MoveAbs(rPosition:= rMovePositionX, rSpeed:= rMoveSpeedX ,rAcceleration:= 0.0, rDeceleration:= 0.0);
		IF stError.ErrorId > 0 THEN
			stError.HardwareGrp := E_HardwareGrp.AxisX;
			nStateA_MoveXY := 99;
		ELSE
			stError.ErrorId := pYDrive^.M_MoveAbs(rPosition:= rMovePositionY, rSpeed:= rMoveSpeedY ,rAcceleration:= 0.0, rDeceleration:= 0.0);
			IF stError.ErrorId > 0 THEN //XDrive muss abgebrochen werden
				pXDrive^.M_Stop();
				stError.HardwareGrp := E_HardwareGrp.AxisY;
				nStateA_MoveXY := 99;
			END_IF
		END_IF
	ELSIF eMoveMode = E_MoveMode.MODE_Home THEN	//auf 0 fahren
		stError.ErrorId := pXDrive^.M_MoveAbs(rPosition:= 0.0, rSpeed:= rMoveSpeedX ,rAcceleration:= 0.0, rDeceleration:= 0.0);
		IF stError.ErrorId > 0 THEN
			stError.HardwareGrp := E_HardwareGrp.AxisX;
			nStateA_MoveXY := 99;
		ELSE
			stError.ErrorId := pYDrive^.M_MoveAbs(rPosition:= 0.0, rSpeed:= rMoveSpeedY ,rAcceleration:= 0.0, rDeceleration:= 0.0);
			IF stError.ErrorId > 0 THEN //XDrive muss abgebrochen werden
				pXDrive^.M_Stop();
				stError.HardwareGrp := E_HardwareGrp.AxisY;
				nStateA_MoveXY := 99;
			END_IF
		END_IF
	END_IF
//Warten bis Positionierung fertig
ELSIF nStateA_MoveXY = 3 THEN
	IF pXDrive^.P_bError THEN
		pYDrive^.M_Stop();
		stError.ErrorId := pXDrive^.P_nErrorId;
		stError.HardwareGrp := E_HardwareGrp.AxisX;
		stError.HardwareNr	:= 1;
		nStateA_MoveXY := 99;
	ELSIF pYDrive^.P_bError THEN
		pXDrive^.M_Stop();
		stError.ErrorId := pYDrive^.P_nErrorId;
		stError.HardwareGrp := E_HardwareGrp.AxisY;
		stError.HardwareNr	:= 1;
		nStateA_MoveXY := 99;
	ELSE
		IF NOT (pXDrive^.P_bBusy OR pYDrive^.P_bBusy) THEN
			nStateA_MoveXY := 80;
		END_IF
	END_IF
//Stoppen
ELSIF nStateA_MoveXY = 70 THEN
	pXDrive^.M_Stop();
	pYDrive^.M_Stop();
	IF NOT (pXDrive^.P_bBusy OR pYDrive^.P_bBusy) THEN
		nStateA_MoveXY := 80;
	END_IF
END_IF

//Errorhandling
IF nStateA_MoveXY = 99 THEN
	stError.ObjectId := nObjectID;
	stError.Cmd := E_Action.ACTION_MoveXY;
	stError.POU := E_POU.POU_FB_MzBase;
	stError.POUAction := E_POUACT.POUACT_A_MoveXY;
	fbErrorList.M_Add(stError);
END_IF
END_ACTION

ACTION A_MoveY:
stError.POUState := nStateA_MoveY;

CASE nStateA_MoveY OF
	0:
		IF NOT bIgnoreZCollision THEN
			//Distanz ermitteln, für ev. Freifahren der Z-Achsen
			IF eMoveMode = E_MoveMode.MODE_Relative THEN
				rDistanceY := rMovePositionY;
			ELSIF eMoveMode = E_MoveMode.MODE_AbsWithOffset THEN
				st3DPoint := P_stCurrentPosTotal;
				rDistanceY := ABS(rMovePositionY - st3DPoint.Y);
			ELSIF eMoveMode = E_MoveMode.MODE_AbsNoneOffset THEN
				rDistanceY := ABS(rMovePositionY - pYDrive^.P_rActPos);
			END_IF
			
			stActionData.eAction := E_Action.ACTION_MoveZ;
			stActionData.aParams[1] := E_MoveMode.MODE_Free;
			stActionData.aParams[3] := -1;	//MaxSpeed
			
			//MoveY erfordert nur, dass die Achsen am selben Head OK sind
			nStateA_MoveY := 1;
			IF NOT P_pMzHead^.P_bCollFree THEN
				stError.ErrorId := P_pMzHead^.M_ExeAction(stActionData);
				IF stError.ErrorId > 0 THEN
					stError.Cmd := E_Action.ACTION_MoveZ;
					nStateA_MoveY := 99;
				END_IF
			END_IF
		ELSE
			nStateA_MoveY := 2;		
		END_IF		

	1:	//warten bis alle Achsen fertig
		nStateA_MoveY := 2;
		pHead := P_pMzHead;
		IF pHead^.M_CheckChildsForActionBusy(E_Action.ACTION_MoveZ) THEN
			nStateA_MoveY := 1;
		END_IF
		
		stError.ErrorId := pHead^.M_CheckChildsForError(); 
		IF stError.ErrorId > 0 THEN
			nStateA_MoveY := 99;
		END_IF

	2:	//In Abhängigkeit von MoveMode absolut oder relativ fahren
		IF eMoveMode = E_MoveMode.MODE_Relative THEN	//Relativ
			stError.ErrorId := pYDrive^.M_MoveRel(rDistance:= rMovePositionY, rSpeed:= rMoveSpeedY, rAcceleration:= 0.0, rDeceleration:= 0.0);
			nStateA_MoveY := 3; 
		ELSIF eMoveMode = E_MoveMode.MODE_AbsWithOffset THEN	//Absolut mit Offsets
			//Achsenposition berechnen
			//Position ergibt sich aus Zielposition abzüglich aller Offsets
			st3DPoint := P_stAbsPosTotal;	//Summe aller Offsets
			rMovePositionY := rMovePositionY - st3DPoint.Y;
			stError.ErrorId := pYDrive^.M_MoveAbs(rPosition:= rMovePositionY, rSpeed:= rMoveSpeedY, rAcceleration:= 0.0, rDeceleration:= 0.0);
			nStateA_MoveY := 3; 
		ELSIF eMoveMode = E_MoveMode.MODE_AbsNoneOffset THEN	//Absolut OHNE Offsets!!
			stError.ErrorId := pYDrive^.M_MoveAbs(rPosition:= rMovePositionY, rSpeed:= rMoveSpeedY, rAcceleration:= 0.0, rDeceleration:= 0.0); 
			nStateA_MoveY := 3;
		ELSIF eMoveMode = E_MoveMode.MODE_Home THEN	//auf 0 fahren
			stError.ErrorId := pYDrive^.M_MoveAbs(rPosition:= 0.0, rSpeed:= rMoveSpeedY, rAcceleration:= 0.0, rDeceleration:= 0.0); 
			nStateA_MoveY := 3;
		ELSE
			nStateA_MoveY := 99; //Error (Dieser Fall sollte nicht auftreten. MoveMode wird in M_ExeAction() abgefangen)
		END_IF
		
		IF stError.ErrorId > 0 THEN
			nStateA_MoveY := 99;
		END_IF	

	3:	//Warten bis Positionierung fertig
		IF NOT pYDrive^.P_bBusy THEN
			IF pYDrive^.P_bError THEN
				stError.ErrorId := pYDrive^.P_nErrorId;
				//fbYDrive resetten!!
 				nStateA_MoveY := 99;
			ELSE
				nStateA_MoveY := 80;
			END_IF
		END_IF

	70:	//Stoppen
		pYDrive^.M_Stop();
		IF NOT pYDrive^.P_bBusy THEN
			nStateA_MoveY := 80;
		END_IF		
END_CASE

//Errorhandling
IF nStateA_MoveY = 99 THEN
	stError.HardwareGrp := E_HardwareGrp.AxisY;
	stError.HardwareNr := 1;
	stError.Cmd := E_Action.ACTION_MoveY;
	stError.POU := E_POU.POU_FB_MzBase;
	stError.POUAction := E_POUACT.POUACT_A_MoveY;
	fbErrorList.M_Add(stError);
END_IF
END_ACTION

ACTION A_MoveZ:

END_ACTION

ACTION A_Reset:
IF nStateA_ResetBase = 0 THEN //ist noch irgendeine Action aktiv?		
	IF bJogXY THEN
		bJogXY := FALSE;
		nStateA_JogXY := 0;
	END_IF
	IF bMoveX THEN
		bMoveX := FALSE;
		bXYIsMoving := FALSE;
		nStateA_MoveX := 0;
	END_IF
	IF bMoveY THEN
		bMoveY := FALSE;
		bXYIsMoving := FALSE;
		nStateA_MoveY := 0;
	END_IF		
	IF bMoveXY THEN
		bMoveXY := FALSE;
		bXYIsMoving := FALSE;
		nStateA_MoveXY := 0;
	END_IF
	IF bMoveZ THEN
		bMoveZ := FALSE;
		nStateA_MoveZ := 80;
	END_IF		
	nStateA_InitAxis := 0;
	nStateA_JogXY := 0;
	nStateA_Stop := 0;
	nStateA_MoveX := 0;
	nStateA_MoveY := 0;
	nStateA_MoveXY := 0;
	nStateA_MoveZ := 0;
	nStateA_ResetBase := 0;
	nStateA_ResetSpec := 0;
	bXYIsMoving := FALSE;
	bZIsMoving := FALSE;		
	nStateA_ResetBase := 1;
ELSIF nStateA_ResetBase = 1 THEN //Warten, bis Drives zurückgesetzt
	IF NOT (pXDrive^.P_bError OR pYDrive^.P_bError) THEN 
		nStateA_ResetBase := 2;
	END_IF
ELSIF nStateA_ResetBase = 2 THEN	//ResetTool ready?		
	IF nStateA_ResetTool = 80 THEN
		stError.ErrorId := 0;
		nStateA_ResetBase := 80;
	ELSIF nStateA_ResetTool >= 80 THEN
		nStateA_ResetBase := 99;
	END_IF
END_IF
END_ACTION

ACTION A_Stop:
//Diese Aktion wird in der Regel vom "FB_Tool.A_stop()" aufgerufen
//kommt der Aufruf von "FB_Tool.A_stop()" das erst mal, ist "nStateA_Stop" = 2

IF nStateA_Stop <= 2 THEN
	IF bInitAxis AND nStateA_InitAxis < 70 THEN
		nStateA_InitAxis := 70;
	END_IF
	
	IF bJogXY AND nStateA_JogXY < 4 THEN
		nStateA_JogXY := 4;
	END_IF
	
	IF bMoveX AND nStateA_MoveX < 70 THEN	//X-Move stoppen
		nStateA_MoveX := 70;
	END_IF
	
	IF bMoveY AND nStateA_Movey < 70 THEN	//X-Move stoppen
		nStateA_MoveY := 70;
	END_IF	
	
	IF bMoveXY AND nStateA_MoveXY < 70 THEN	//X-Move stoppen
		bFlagMoveX := TRUE;
		bFlagMoveY := TRUE;
		nStateA_MoveXY := 70;
	END_IF

	IF bMoveZ AND nStateA_MoveZ < 70 THEN	//Z-Move stoppen
		nStateA_MoveZ := 70;
	END_IF
	
	nStateA_Stop := 3;

ELSIF nStateA_Stop = 3 THEN
	//Warten bis alle Actions abgebrochen
	IF hList.nCount = 1 THEN	//nur der Eintrag von Stop
		nStateA_Stop := 80;
	END_IF	
END_IF
END_ACTION

METHOD M_AddChild : ERRORID
VAR_INPUT
	pObject	: POINTER TO FB_Object;
	nSlotNr	: UINT;
	nIndex : INT;
END_VAR
//Die Methode muss zwingend von den abgeleiteten FBs implementiert werden
END_METHOD

METHOD M_CancelAction
VAR_INPUT
	eAction : E_Action;
END_VAR
CASE eAction OF
	E_Action.ACTION_Init:
		IF bInitAxis AND nStateA_InitAxis < 70 THEN
			nStateA_InitAxis := 70;
		END_IF	
	E_Action.ACTION_Jog:
		IF bJogXY AND nStateA_JogXY < 4 THEN	//Jogging stoppen
			nStateA_JogXY := 4;
		END_IF	
	E_Action.ACTION_MoveX:
		IF bMoveX AND nStateA_MoveX < 70 THEN	//X-Move stoppen
			nStateA_MoveX := 70;
		END_IF	
	E_Action.ACTION_MoveY:
		IF bMoveY AND nStateA_Movey < 70 THEN	//X-Move stoppen
			nStateA_MoveY := 70;
		END_IF	
	E_Action.ACTION_MoveZ:
		IF bMoveZ AND nStateA_MoveZ < 70 THEN	//Z-Move stoppen
			nStateA_MoveZ := 70;
		END_IF	
	E_Action.ACTION_MoveXY:
		IF bMoveXY AND nStateA_MoveXY < 70 THEN	//X-Move stoppen
			bFlagMoveX := TRUE;
			bFlagMoveY := TRUE;
			nStateA_MoveXY := 70;
		END_IF
END_CASE
END_METHOD

METHOD M_CheckAction : ERRORID
VAR_INPUT
	refActionData 	: REFERENCE TO ST_ActionData;
	pCorrelObject	: POINTER TO FB_Object;
END_VAR
M_CheckAction := E_ErrorIdCmd.ERRORID_InvalidAction;
END_METHOD

METHOD M_CheckMoveLimit : BOOL
VAR_INPUT
	sAxis			: STRING[2];
	eMoveMode		: E_MoveMode;
	rMovePosition	: REAL;
END_VAR

VAR
	st3DPoint		: ST_3DPoint;
	rMovePosTemp	: REAL;
END_VAR
IF sAxis = 'X' THEN 
	IF eMoveMode = E_MoveMode.MODE_Relative THEN	//Relativ
		rMovePosTemp := pXDrive^.P_rActPos + rMovePosition; 
	ELSIF eMoveMode = E_MoveMode.MODE_AbsWithOffset THEN	//Absolut mit Offsets
		st3DPoint := P_stAbsPosTotal;	//Summe aller Offsets
		rMovePosTemp := rMovePosition - st3DPoint.X;
	ELSIF eMoveMode = E_MoveMode.MODE_AbsNoneOffset THEN	//Absolut OHNE Offsets!!
		rMovePosTemp := rMovePosition;
	END_IF
	
	IF rMovePosTemp >= pXDrive^.P_rMinPos AND rMovePosTemp <= pXDrive^.P_rMaxPos THEN
		M_CheckMoveLimit := TRUE;
	END_IF
ELSIF sAxis = 'Y' THEN
	IF eMoveMode = E_MoveMode.MODE_Relative THEN	//Relativ
		rMovePosTemp := pYDrive^.P_rActPos + rMovePosition; 
	ELSIF eMoveMode = E_MoveMode.MODE_AbsWithOffset THEN	//Absolut mit Offsets
		st3DPoint := P_stAbsPosTotal;	//Summe aller Offsets
		rMovePosTemp := rMovePosition - st3DPoint.Y;
	ELSIF eMoveMode = E_MoveMode.MODE_AbsNoneOffset THEN	//Absolut OHNE Offsets!!
		rMovePosTemp := rMovePosition;
	END_IF

	IF rMovePosTemp >= pYDrive^.P_rMinPos AND rMovePosTemp <= pYDrive^.P_rMaxPos THEN
		M_CheckMoveLimit := TRUE;
	END_IF
END_IF
END_METHOD

METHOD M_CheckProcDataType : BOOL
VAR_INPUT
	eProcDataType : E_ProcDataType;
END_VAR
END_METHOD

METHOD M_CheckProps : ERRORID
VAR_INPUT
END_VAR
END_METHOD

METHOD M_ClearAllProps
VAR_INPUT
	bIgnoreParent : BOOL; //Es wird das gesamte OD gelöscht. -> Zeiger auf Parent nicht mehr gültig!
END_VAR
pPiece := 0;
bInitFB := TRUE;
nObjectID := 0;
nDeviceIdx := 0;
nNotifyId := 0;
fbSlotList.M_Reset();
pObjCollectNode := 0;
MEMSET(ADR(stProcessData),0,SIZEOF(stProcessData));
END_METHOD

METHOD M_ClearOffset
VAR_INPUT
END_VAR
stOffset.X := 0.0;
stOffset.Y := 0.0;
stOffset.Z := 0.0;
END_METHOD

METHOD M_ExeAction : ERRORID
VAR_INPUT
	refActionData : REFERENCE TO ST_ActionData;	
END_VAR
VAR
	bRiskOfCrash	: BOOL;
END_VAR
//In dieser Methode muss gecheckt werden, ob die entsprechende BasicAction auch zum aktuellen Zeitpunkt auch ausgeführt werden kann
bCanceled := FALSE;	//wozu das ??

IF NOT (eCurrentState = E_MachineState.MACHINESTATE_Idle OR
	eCurrentState = E_MachineState.MACHINESTATE_Active OR
	eCurrentState = E_MachineState.MACHINESTATE_Ready) THEN
	M_ExeAction := E_ErrorIdCmd.ERRORID_InvalidState;
	RETURN;
END_IF

CASE refActionData.eAction OF
	E_Action.ACTION_Init:
		IF NOT bInitAxis THEN
			bReInit := DINT_TO_BOOL(refActionData.aParams[1]);
			bInitAxis := TRUE;			
			fbList.A_AddHeadValue(hList := hList, putValue := E_Action.ACTION_Init); 
			//bIsInit := FALSE;
		ELSE
			RETURN;
		END_IF
		
	E_Action.ACTION_Jog:
		
		//XY-Axis muss initialisiert sein
		//Wenn kein MzHead, dann fragen, ob übergeordneter MzHead initialisiert
		IF NOT P_bXYIsInit THEN
			M_ExeAction := E_ErrorIdCmd.ERRORID_DeviceNotInitialized;
			RETURN;
		END_IF
		//Action darf eingetragen werden wenn:
		//wenn Action noch nicht aktiv oder
		//wenn Action aktiv und nJogDirection = 0
		//wenn Action aktiv und Jogmode = Continous und aktueller Jogmode = Continous

		eJogXYDirectionNew := DINT_TO_USINT(refActionData.aParams[2]);
		bJogXYModeInchingNew := DINT_TO_BOOL(refActionData.aParams[1]);
		//rJogXYSpeed wird weiter unten in Abhängigkeit von Richtung gesetzt
		
		rJogXYDistance := DINT_TO_REAL(refActionData.aParams[4]);
		
		//Wenn es einen Richtungswechsel gibt, dann darf "bJogXY" nicht aktiv sein
		
		IF bJogXY THEN //Action schon aktiv 
			//Wird nur ausgeführt wenn:
			//JogDirection = E_MoveDirection.DIRECTION_STOP
			//neuer und alter JogMode = Continous
			IF NOT ((eJogXYDirectionNew = E_MoveDirection.DIRECTION_STOP) OR 
					((eJogXYDirectionNew = eJogXYDirection) AND
					(bJogXYModeInchingNew = FALSE AND bJogXYModeInching = FALSE))) THEN
				RETURN;
			END_IF
		ELSE
			IF eJogXYDirectionNew = E_MoveDirection.DIRECTION_XPLUS OR eJogXYDirectionNew = E_MoveDirection.DIRECTION_XMINUS
 				OR eJogXYDirectionNew = E_MoveDirection.DIRECTION_YPLUS OR eJogXYDirectionNew = E_MoveDirection.DIRECTION_YMINUS THEN
				//Checken ob bei im Inching-Mode die Endlagen überschritten werden
				IF bJogXYModeInchingNew THEN	//Inching-Mode
					CASE eJogXYDirectionNew OF
						E_MoveDirection.DIRECTION_XPLUS:
							IF (pXDrive^.P_rActPos + rJogXYDistance) > pXDrive^.P_rMaxPos THEN
								rJogXYDistance := pXDrive^.P_rMaxPos - pXDrive^.P_rActPos - 5.0;
							END_IF
						E_MoveDirection.DIRECTION_XMINUS:
							IF (pXDrive^.P_rActPos - rJogXYDistance) < pXDrive^.P_rMinPos THEN
								//JogDistance auf aktuelle Distance - 5 verkleinern
								rJogXYDistance := pXDrive^.P_rActPos - pXDrive^.P_rMinPos;
								IF rJogXYDistance < 0.0 THEN
									rJogXYDistance := 0.0;
								END_IF
							END_IF
						E_MoveDirection.DIRECTION_YPLUS:
							IF (pYDrive^.P_rActPos + rJogXYDistance) > pYDrive^.P_rMaxPos THEN
								rJogXYDistance := pYDrive^.P_rMaxPos - pYDrive^.P_rActPos - 5.0;
							END_IF
						E_MoveDirection.DIRECTION_YMINUS:
							IF (pYDrive^.P_rActPos - rJogXYDistance) < pYDrive^.P_rMinPos THEN
								rJogXYDistance := pYDrive^.P_rActPos - 5.0;
							END_IF
					END_CASE
				END_IF
				//Checken ob MzTools kollisionsfrei und Speed setzen
				IF eJogXYDirectionNew = E_MoveDirection.DIRECTION_YPLUS OR eJogXYDirectionNew = E_MoveDirection.DIRECTION_YMINUS THEN
					rJogXYSpeed := MIN(DINT_TO_REAL(refActionData.aParams[3]),pYDrive^.P_rMaxSpeed);
					IF NOT P_pMzHead^.P_bCollFree THEN
						bRiskOfCrash := TRUE;
					END_IF
				ELSIF eJogXYDirectionNew = E_MoveDirection.DIRECTION_XPLUS OR eJogXYDirectionNew = E_MoveDirection.DIRECTION_XMINUS THEN
					rJogXYSpeed := MIN(DINT_TO_REAL(refActionData.aParams[3]),pXDrive^.P_rMaxSpeed);
					//Hier muss die Kollisionsgefährung aller Köpfe gecheckt werden
					FOR i:= 1 TO fbObjectDirectory.nCntMZHead BY 1 DO
						IF NOT afbMzHead[i].P_bCollFree THEN
							bRiskOfCrash := TRUE;
						END_IF
					END_FOR
				END_IF
				
				IF bRiskOfCrash THEN
					IF bJogXYModeInchingNew THEN	//Modus Inching -> nur Schrittweite von max 1mm zulassen
						IF rJogXYDistance > 1000.0 THEN
							M_ExeAction := E_ErrorIdCmd.ERRORID_JogDistanceRiskOfCrash;
							RETURN;
						END_IF
					ELSE	//Modus Continous -> nur Geschwindigkeit von max 1mm/sec
						IF rJogXYSpeed > 5000.0 THEN
							M_ExeAction := E_ErrorIdCmd.ERRORID_JogSpeedRiskOfCrash;
							RETURN;
						END_IF
					END_IF
				END_IF
			ELSE
				IF NOT bJogXYModeInchingNew THEN
					rJogXYDistance := 999999.9;
				END_IF
			END_IF
		END_IF

		eJogXYDirection := eJogXYDirectionNew;
		bJogXYModeInching := bJogXYModeInchingNew;
		
		//In LinkedListCtrl eintragen - wenn schon vorhanden, dann überschreiben!!
		getPosPtr := 0;	//nach vorhandenem Eintrag suchen - beginnen an Anfang
		fbList.A_FindNext(hList := hList, putPosPtr := getPosPtr, putValue := E_Action.ACTION_Jog, getValue=>getValue, getPosPtr=>getPosPtr );

		IF NOT fbList.bOk THEN	//Eintrag wurde nicht gefunden
			//Übeprüfen, ob jeweilige Achse referenziert
			IF eJogXYDirection = E_MoveDirection.DIRECTION_XPLUS OR eJogXYDirection = E_MoveDirection.DIRECTION_XMINUS THEN	//X
				IF NOT pXDrive^.P_bHomed THEN
					M_ExeAction := E_ErrorIdMultiZ.ERRORID_AxisNotHomed;
					RETURN;
				END_IF
			ELSIF eJogXYDirection = E_MoveDirection.DIRECTION_YPLUS OR eJogXYDirection = E_MoveDirection.DIRECTION_YMINUS THEN	//Y
				IF NOT pYDrive^.P_bHomed THEN
					M_ExeAction := E_ErrorIdMultiZ.ERRORID_AxisNotHomed;
					RETURN;
				END_IF
			END_IF
			bJogXY := TRUE;
			bJogXYImpuls := TRUE;
			bJogXYClock := TRUE;			
			fbList.A_AddHeadValue(hList := hList, putValue := E_Action.ACTION_Jog);
			bBusy := TRUE;
		ELSE	//Eintrag wurde gefunden
			bJogXYClock := NOT bJogXYClock;
			bJogXYImpuls := TRUE;
		END_IF
	
	E_Action.ACTION_MoveX:
		IF NOT bMoveX THEN 
			IF NOT pXDrive^.P_bHomed THEN
				M_ExeAction := E_ErrorIdMultiZ.ERRORID_AxisNotHomed;
				RETURN;
			END_IF
			
			//Check MoveMode			
			eMoveMode := DINT_TO_USINT(refActionData.aParams[1]);
			IF NOT (eMoveMode = E_MoveMode.MODE_Relative OR eMoveMode = E_MoveMode.MODE_AbsWithOffset OR
				eMoveMode = E_MoveMode.MODE_AbsWithOffset OR eMoveMode = E_MoveMode.MODE_AbsNoneOffset OR
 				eMoveMode = E_MoveMode.MODE_Home) THEN
				M_ExeAction := E_ErrorIdCmd.ERRORID_InvalidMoveMode;  //Error
				RETURN;			
			END_IF
			
			rMovePositionX := DINT_TO_REAL(refActionData.aParams[2]);
			//Targetposition auf Limits checken
			IF NOT M_CheckMoveLimit(sAxis:= 'X', eMoveMode:= eMoveMode,rMovePosition:= rMovePositionX) THEN
				M_ExeAction := E_ErrorIdCmd.ERRORID_TargetPosOutOfRangeX;  //Error
				RETURN;
			END_IF

			rMoveSpeedX := MIN(DINT_TO_REAL(refActionData.aParams[3]),pXDrive^.P_rMaxSpeed);
			
			IF rMoveSpeedX < 0 THEN //Geschwindigkeitsangabe -1 = max. Geschwindigkeit
				rMoveSpeedX := pXDrive^.P_rMaxSpeed;
			END_IF
			
			bIgnoreZCollision := DINT_TO_BOOL(refActionData.aParams[4]);
			bMoveXReady := FALSE;
			bXYIsMoving := TRUE;
			bMoveX := TRUE;
			fbList.A_AddHeadValue(hList := hList, putValue := E_Action.ACTION_MoveX);
		ELSE
			M_ExeAction := E_ErrorIdCmd.ERRORID_BasicActionActive;  //Error
			RETURN;			
		END_IF
		
	E_Action.ACTION_MoveY:
		IF NOT bMoveY THEN
			IF NOT pYDrive^.P_bHomed THEN
				M_ExeAction := E_ErrorIdMultiZ.ERRORID_AxisNotHomed;
				RETURN;
			END_IF
			
			//Check MoveMode			
			eMoveMode := DINT_TO_USINT(refActionData.aParams[1]);
			IF NOT (eMoveMode = E_MoveMode.MODE_Relative OR eMoveMode = E_MoveMode.MODE_AbsWithOffset OR
				eMoveMode = E_MoveMode.MODE_AbsWithOffset OR eMoveMode = E_MoveMode.MODE_AbsNoneOffset OR
 				eMoveMode = E_MoveMode.MODE_Home) THEN
				M_ExeAction := E_ErrorIdCmd.ERRORID_InvalidMoveMode;  //Error
				RETURN;			
			END_IF			

			rMovePositionY := DINT_TO_REAL(refActionData.aParams[2]);
			//Targetposition auf Limits checken
			IF NOT M_CheckMoveLimit(sAxis:= 'Y', eMoveMode:= eMoveMode,rMovePosition:= rMovePositionY) THEN
				M_ExeAction := E_ErrorIdCmd.ERRORID_TargetPosOutOfRangeY;
				RETURN;
			END_IF
			
			rMoveSpeedY := MIN(DINT_TO_REAL(refActionData.aParams[3]),pYDrive^.P_rMaxSpeed);
			
			IF rMoveSpeedY < 0 THEN //Geschwindigkeitsangabe -1 = max. Geschwindigkeit
				rMoveSpeedY := pYDrive^.P_rMaxSpeed;
			END_IF
			
			bIgnoreZCollision := DINT_TO_BOOL(refActionData.aParams[4]);			
			bMoveYReady := FALSE;
			bXYIsMoving := TRUE;
			bMoveY := TRUE;							
			fbList.A_AddHeadValue(hList := hList, putValue := E_Action.ACTION_MoveY);
		ELSE
			M_ExeAction := E_ErrorIdCmd.ERRORID_BasicActionActive;  //Error
			RETURN;			
		END_IF
	
	E_Action.ACTION_MoveXY:	
		IF NOT bMoveXY THEN
			IF NOT (pXDrive^.P_bHomed AND pYDrive^.P_bHomed) THEN
				M_ExeAction := E_ErrorIdMultiZ.ERRORID_AxisNotHomed;
				RETURN;
			END_IF
			
			//Check MoveMode			
			eMoveMode := DINT_TO_USINT(refActionData.aParams[1]);
			IF NOT (eMoveMode = E_MoveMode.MODE_Relative OR eMoveMode = E_MoveMode.MODE_AbsWithOffset OR
				eMoveMode = E_MoveMode.MODE_AbsWithOffset OR eMoveMode = E_MoveMode.MODE_AbsNoneOffset OR
 				eMoveMode = E_MoveMode.MODE_Home) THEN
				M_ExeAction := E_ErrorIdCmd.ERRORID_InvalidMoveMode;  //Error
				RETURN;			
			END_IF			

			//Targetposition X auf Limits checken
			rMovePositionX := DINT_TO_REAL(refActionData.aParams[2]);
			IF NOT M_CheckMoveLimit(sAxis:= 'X', eMoveMode:= eMoveMode,rMovePosition:= rMovePositionX) THEN
				M_ExeAction := E_ErrorIdCmd.ERRORID_TargetPosOutOfRangeX;
				RETURN;
			END_IF
			
			//Targetposition Y auf Limits checken
			rMovePositionY := DINT_TO_REAL(refActionData.aParams[3]);
			IF NOT M_CheckMoveLimit(sAxis:= 'Y', eMoveMode:= eMoveMode,rMovePosition:= rMovePositionY) THEN
				M_ExeAction := E_ErrorIdCmd.ERRORID_TargetPosOutOfRangeY;
				RETURN;
			END_IF
			
			rMoveSpeedX := MIN(DINT_TO_REAL(refActionData.aParams[4]),pXDrive^.P_rMaxSpeed);
			rMoveSpeedY := MIN(DINT_TO_REAL(refActionData.aParams[5]),pYDrive^.P_rMaxSpeed);
			
			IF rMoveSpeedX < 0 THEN //Geschwindigkeitsangabe -1 = max. Geschwindigkeit
				rMoveSpeedX := pXDrive^.P_rMaxSpeed;
			END_IF

			IF rMoveSpeedY < 0 THEN //Geschwindigkeitsangabe -1 = max. Geschwindigkeit
				rMoveSpeedY := pYDrive^.P_rMaxSpeed;
			END_IF

			eCrashAvoidanceMode := DINT_TO_USINT(refActionData.aParams[6]);
			bSynchron := DINT_TO_BOOL(refActionData.aParams[7]);
			
			bMoveXYReady := FALSE;
			bMoveXReady := FALSE;
			bMoveYReady := FALSE;
			bXYIsMoving := TRUE;
			bMoveXY := TRUE;							
			fbList.A_AddHeadValue(hList := hList, putValue := E_Action.ACTION_MoveXY);
		ELSE
			M_ExeAction := E_ErrorIdCmd.ERRORID_BasicActionActive;  //Error
			RETURN;
		END_IF		
		
	E_Action.ACTION_Stop:
		//Stop braucht nur ausgeführt werden, wenn irgendwas aktiv ist
		IF bBusy AND NOT bStop AND hList.nCount > 0 THEN
			bStop := TRUE;
			fbList.A_AddHeadValue(hList := hList, putValue := E_Action.ACTION_Stop);
		ELSE
			RETURN;
		END_IF
	ELSE
		M_ExeAction := E_ErrorIdCmd.ERRORID_InvalidAction; //Error
		RETURN;
END_CASE

eCurrentState := E_MachineState.MACHINESTATE_Active;
bBusy := TRUE;
END_METHOD

METHOD M_GetActionBusy : BOOL
VAR_INPUT
	eAction : E_Action;
END_VAR
getPosPtr := 0;(* start from first node element *)
fbList.A_FindNext( hList := hList, putPosPtr := getPosPtr, putValue := eAction, getValue=>getValue, getPosPtr=>getPosPtr );
IF fbList.bOk THEN	//Eintrag wurde gefunden, d.h. Action ist noch busy
	M_GetActionBusy := TRUE;
END_IF
END_METHOD

METHOD M_GetAllProps : ERRORID
VAR_INPUT
	refCmdData : REFERENCE TO  ST_CmdData;
END_VAR

VAR
	i 			: UINT;
	pSlot		: POINTER TO FB_Slot;
	stTempPos 	: ST_3DPoint;
END_VAR
refCmdData.aHeader[0] := nObjectID;
refCmdData.aHeader[1] := eObjectType;
refCmdData.aHeader[2]:= nNotifyId;


//Offset lesen
refCmdData.n32Data[2] :=  REAL_TO_DINT(stRelPos.X);
refCmdData.n32Data[3] :=  REAL_TO_DINT(stRelPos.Y);
refCmdData.n32Data[4] :=  REAL_TO_DINT(stRelPos.Z);
//Offset1 lesen
refCmdData.n32Data[5] :=  REAL_TO_DINT(stOffset.X);
refCmdData.n32Data[6] :=  REAL_TO_DINT(stOffset.Y);
refCmdData.n32Data[7] :=  REAL_TO_DINT(stOffset.Z);

refCmdData.n32Data[8] :=  nNumberOfSlots;

nCurrentPropIndex := 8;

fbSlotList.M_SetCurrentToHead();

FOR i := 1 TO nNumberOfSlots BY 1 DO
	pSlot := fbSlotList.M_GetNext();
	IF pSlot > 0 THEN
		nCurrentPropIndex := nCurrentPropIndex + 1;
		refCmdData.n32Data[nCurrentPropIndex] := pSlot^.P_nNr;
		stTempPos := pSlot^.P_stRelPos;
		nCurrentPropIndex := nCurrentPropIndex + 1;
		refCmdData.n32Data[nCurrentPropIndex] := REAL_TO_DINT(stTempPos.X);
		nCurrentPropIndex := nCurrentPropIndex + 1;
		refCmdData.n32Data[nCurrentPropIndex] := REAL_TO_DINT(stTempPos.Y);
		nCurrentPropIndex := nCurrentPropIndex + 1;
		refCmdData.n32Data[nCurrentPropIndex] := REAL_TO_DINT(stTempPos.Z);		
	END_IF
END_FOR
END_METHOD

METHOD M_GetCollFree : BOOL
VAR_INPUT
	rDistanceX : REAL;
	rDistanceY : REAL;
END_VAR

VAR
	stCurrPos : ST_3DPoint;
	fbRect : FB_Rectangle;
END_VAR
stCurrPos := P_stCurrentPosPhys;
fbRect.X1 := stCurrPos.X;
fbRect.Y1 := stCurrPos.Y;
fbRect.X2 := stCurrPos.X + rDistanceX;
fbRect.Y2 := stCurrPos.Y + rDistanceY;
bDisableFreeMove := FALSE;
IF F_RectInnerRect(fbRect,stAreaCollFree) THEN
	bDisableFreeMove := TRUE;
	M_GetCollFree := TRUE;
ELSIF P_bCollFree THEN
	M_GetCollFree := TRUE;
END_IF
END_METHOD

METHOD M_GetDevice : I_Device
VAR_INPUT
END_VAR
M_GetDevice := THIS^;
END_METHOD

METHOD M_GetFirstErrorChild : POINTER TO FB_MzTool
VAR_INPUT
	bSelf : BOOL;
END_VAR

VAR
	pSlot : POINTER TO FB_Slot;
	pTool : POINTER TO FB_MzTool;
END_VAR
IF bSelf AND P_bError THEN
	M_GetFirstErrorChild := THIS;
	RETURN;
END_IF
fbSlotList.M_SetCurrentToHead();
REPEAT
	pSlot := fbSlotList.M_GetNext();
	IF pSlot > 0 THEN
		IF pSlot^.P_pChild > 0 THEN
			IF pSlot^.P_pChild^.M_bIsGroup(E_ObjectGroup.OBJECTGROUP_MzTool) THEN
				pTool := pSlot^.P_pChild;
				M_GetFirstErrorChild := pTool^.M_GetFirstErrorChild(TRUE);
				IF M_GetFirstErrorChild > 0 THEN
					RETURN;
				END_IF
			END_IF
		END_IF
	END_IF
UNTIL (pSlot = 0)
END_REPEAT
END_METHOD

METHOD M_GetMaxSpeed : REAL
VAR_INPUT
	eDirection : E_MoveDirection;
END_VAR
CASE eDirection OF
	E_MoveDirection.DIRECTION_XMINUS, E_MoveDirection.DIRECTION_XPLUS:
		IF pXDrive > 0 THEN
			M_GetMaxSpeed := pXDrive^.P_rMaxSpeed;
		END_IF
	E_MoveDirection.DIRECTION_YMINUS, E_MoveDirection.DIRECTION_YPLUS:
		IF pYDrive > 0 THEN
			M_GetMaxSpeed := pYDrive^.P_rMaxSpeed;
		END_IF
END_CASE
END_METHOD

METHOD M_GetMinMaxActPos
VAR_INPUT
	pData : POINTER TO ARRAY[0..19] OF DINT;
END_VAR
VAR
	stAbsPosTotal : ST_3DPoint;
END_VAR
MEMSET(pData,0,SIZEOF(pData^));
stAbsPosTotal := P_stAbsPosTotal;
IF pXDrive > 0 THEN
	pData^[0] := REAL_TO_DINT(pXDrive^.P_rMinPos + stAbsPosTotal.X);
	pData^[1] := REAL_TO_DINT(pXDrive^.P_rMaxPos + stAbsPosTotal.X);	
END_IF
IF pYDrive > 0 THEN
	pData^[2] := REAL_TO_DINT(pYDrive^.P_rMinPos + stAbsPosTotal.Y);
	pData^[3] := REAL_TO_DINT(pYDrive^.P_rMaxPos + stAbsPosTotal.Y);	
END_IF

//wird in den abgeleiteten FBs weiter verrechnet
pData^[4] := REAL_TO_DINT(stAbsPosTotal.Z);
pData^[5] := pData^[4];
END_METHOD

METHOD M_GetProcData : DINT
VAR_INPUT
	eProcDataType : E_ProcDataType;
END_VAR
END_METHOD

METHOD M_GetPropCheckSum : UINT
VAR_INPUT
END_VAR

VAR
	i			: UINT;
	stData 		: ST_CmdData;
END_VAR
M_GetAllProps(stData);
wChecksum := F_DATA_TO_CRC16_CCITT(ADR(stData.n32Data[0]),nNoOfProps * 4,16#FFFF);
M_GetPropCheckSum := wChecksum;
END_METHOD

METHOD M_GetSlot : POINTER TO FB_Slot
VAR_INPUT
	nSlotNr	: UINT;
END_VAR
M_GetSlot := fbSlotList.M_GetAtNr(nSlotNr);
END_METHOD

METHOD M_GetSlotFromChild : POINTER TO FB_Slot
VAR_INPUT
	pObject : POINTER TO FB_Object;
END_VAR

VAR
	pSlot : POINTER TO FB_Slot;
END_VAR
//Die SlotList iterieren und vergleichen ob Objekte übereinstimmen
fbSlotList.M_SetCurrentToHead();
REPEAT
	pSlot := fbSlotList.M_GetNext();
	IF pSlot > 0 THEN
		IF pSlot^.P_pChild = pObject THEN
			M_GetSlotFromChild := pSlot;
			EXIT;
		END_IF
	END_IF
UNTIL pSlot = 0
END_REPEAT
END_METHOD

METHOD M_GetXYRange : ST_Rectangle
VAR_INPUT
END_VAR
VAR
	stAbsPosTotal : ST_3DPoint;
END_VAR
stAbsPosTotal := P_stAbsPosTotal;
IF pXDrive > 0 THEN
	M_GetXYRange.X1 := pXDrive^.P_rMinPos + stAbsPosTotal.X;
	M_GetXYRange.X2 := pXDrive^.P_rMaxPos + stAbsPosTotal.X;	
END_IF
IF pYDrive > 0 THEN
	M_GetXYRange.Y1 := pYDrive^.P_rMinPos + stAbsPosTotal.Y;
	M_GetXYRange.Y2 := pYDrive^.P_rMaxPos + stAbsPosTotal.Y;	
END_IF
END_METHOD

METHOD M_GetZAxisRef : POINTER TO FB_ZAxisRef
VAR_INPUT
	pTool : POINTER TO FB_MzTool;
	pToolSlot : POINTER TO FB_Slot;
END_VAR
END_METHOD

METHOD M_RawPosToRealPos : ST_3DPoint
VAR_INPUT
	stRawPos : ST_3DPoint;
END_VAR

VAR
	stTemp		: ST_3DPoint;
	stAbsPos : ST_3DPoint;
END_VAR
END_METHOD

METHOD M_RemoveListEntry : BOOL
VAR_INPUT
	nSearchValue	: E_Action;
END_VAR
getPosPtr := 0;(* start from first node element *)
fbList.A_FindNext( hList := hList, putPosPtr := getPosPtr, putValue := nSearchValue, getValue=>getValue, getPosPtr=>getPosPtr );
IF fbList.bOk THEN	//Eintrag wurde gefunden
	fbList.A_RemoveValueAtPosPtr(hList:= hList,	putPosPtr:= getPosPtr);
	IF fbList.bOk THEN
		M_RemoveListEntry := TRUE;
	END_IF
END_IF
END_METHOD

METHOD M_Reset
bBusy := TRUE;
bFlagA_ResetBase := TRUE;
eCurrentState := E_MachineState.MACHINESTATE_Reset;
END_METHOD

METHOD M_SetAllProps : ERRORID
VAR_INPUT
	refCmdData : REFERENCE TO  ST_CmdData;
END_VAR

VAR
	nMzToolObjId		: UINT;
	nParentMzToolObjId	: UINT;
	i 					: UINT;
	pSlot 				: POINTER TO FB_Slot;
	stTempPos 			: ST_3DPoint;
END_VAR

//RelPos setzen
stRelPos.X:= DINT_TO_REAL(refCmdData.n32Data[2]);
stRelPos.Y:= DINT_TO_REAL(refCmdData.n32Data[3]);
stRelPos.Z:= DINT_TO_REAL(refCmdData.n32Data[4]);
//Offset setzen
stOffset.X:= DINT_TO_REAL(refCmdData.n32Data[5]);
stOffset.Y:= DINT_TO_REAL(refCmdData.n32Data[6]);
stOffset.Z:= DINT_TO_REAL(refCmdData.n32Data[7]);

nCurrentPropIndex := 8;

//Slots parametrieren
nFirstSlotPropIndex := nCurrentPropIndex;
nNumberOfSlots := DINT_TO_UINT(refCmdData.n32Data[nCurrentPropIndex]);

//Falls SlotList noch nicht existiert, dann neue erstellen
IF fbSlotList.P_nCount = 0 THEN
	FOR i:= 1 TO nNumberOfSlots BY 1 DO
		pSlot := __NEW(FB_Slot(pOwner := THIS));
		fbSlotList.M_Add(pSlot);
		nCurrentPropIndex := nCurrentPropIndex + 1;
		pSlot^.P_nNr := DINT_TO_USINT(refCmdData.n32Data[nCurrentPropIndex]);
		nCurrentPropIndex := nCurrentPropIndex + 1;
		stTempPos.X := DINT_TO_REAL(refCmdData.n32Data[nCurrentPropIndex]);
		nCurrentPropIndex := nCurrentPropIndex + 1;
		stTempPos.Y := DINT_TO_REAL(refCmdData.n32Data[nCurrentPropIndex]);
		nCurrentPropIndex := nCurrentPropIndex + 1;
		stTempPos.Z := DINT_TO_REAL(refCmdData.n32Data[nCurrentPropIndex]);
		pSlot^.P_stRelPos := stTempPos;
	END_FOR
ELSE
	IF nNumberOfSlots <> fbSlotList.P_nCount THEN
		M_SetAllProps := E_ErrorIdObjMgmt.ERRORID_ChangeNoOfSlotsNotAllowed;
		RETURN;
	END_IF
	FOR i:= 1 TO nNumberOfSlots BY 1 DO
		nCurrentPropIndex := nCurrentPropIndex + 1;
		pSlot := fbSlotList.M_GetAtNr(DINT_TO_USINT(refCmdData.n32Data[nCurrentPropIndex]));
		IF pSlot > 0 THEN
			nCurrentPropIndex := nCurrentPropIndex + 1;
			stTempPos.X := DINT_TO_REAL(refCmdData.n32Data[nCurrentPropIndex]);
			nCurrentPropIndex := nCurrentPropIndex + 1;
			stTempPos.Y := DINT_TO_REAL(refCmdData.n32Data[nCurrentPropIndex]);
			nCurrentPropIndex := nCurrentPropIndex + 1;
			stTempPos.Z := DINT_TO_REAL(refCmdData.n32Data[nCurrentPropIndex]);
			pSlot^.P_stRelPos := stTempPos;
		ELSE
			M_SetAllProps := 222;
			RETURN;
		END_IF
	END_FOR
END_IF
nLastSlotPropIndex := nCurrentPropIndex;

nNoOfProps := nCurrentPropIndex + 1;
END_METHOD

METHOD M_SetSingleProp : ERRORID
VAR_INPUT
	refCmdData : REFERENCE TO  ST_CmdData;
END_VAR

VAR
	nSlotIndex	: UINT;
	nIndex		: UINT;
	pSlot		: POINTER TO FB_Slot;
END_VAR
//Basisproperties schreiben
CASE refCmdData.aHeader[1] OF	//Property-Nr
	2:	//RelPosX
		stRelPos.X := DINT_TO_REAL(refCmdData.n32Data[0]);
	3:	//RelPosY
		stRelPos.Y := DINT_TO_REAL(refCmdData.n32Data[0]);
	4:	//RelPosZ
		stRelPos.Z := DINT_TO_REAL(refCmdData.n32Data[0]);
	5:	//OffsetY
		stOffset.X := DINT_TO_REAL(refCmdData.n32Data[0]);
	6:	//OffsetY
		stOffset.Y := DINT_TO_REAL(refCmdData.n32Data[0]);
	7:	//OffsetY
		stOffset.Z := DINT_TO_REAL(refCmdData.n32Data[0]);
	8:	//NumberOfSlots
		M_SetSingleProp := E_ErrorIdCmd.ERRORID_InvalidProperty;
	ELSE
		//Handelt es sich bei dem PropNr um eine SlotPropNr?
		IF refCmdData.aHeader[1] >= nFirstSlotPropIndex AND refCmdData.aHeader[1] <= nLastSlotPropIndex THEN
			nIndex := (refCmdData.aHeader[1]- nFirstSlotPropIndex);	
			IF nIndex MOD 4 = 0 THEN
				nSlotIndex := nIndex / 4;
			ELSE
				nSlotIndex := nIndex / 4 + 1;
			END_IF		
			pSlot := fbSlotList.M_GetAtIndex(nSlotIndex);
			IF pSlot > 0 THEN
				nIndex := nIndex - ((nSlotIndex - 1)* 4);
				CASE nIndex OF
					2:	pSlot^.P_rRelPosX := DINT_TO_REAL(refCmdData.n32Data[0]);
					
					3:	pSlot^.P_rRelPosY := DINT_TO_REAL(refCmdData.n32Data[0]);
					
					4:	pSlot^.P_rRelPosZ := DINT_TO_REAL(refCmdData.n32Data[0]);
				END_CASE
			END_IF			
		ELSE
			M_SetSingleProp := E_ErrorIdCmd.ERRORID_InvalidProperty;
		END_IF
END_CASE
END_METHOD

METHOD M_Stop : ERRORID
VAR_INPUT
END_VAR
stActionData.eAction := E_Action.ACTION_Stop;
M_ExeAction(stActionData);
END_METHOD

METHOD M_UpdateParent
VAR_INPUT
END_VAR
END_METHOD

PROPERTY P_bBusy : BOOL
GET
P_bBusy := bBusy;
END_GET
END_PROPERTY

PROPERTY P_bCanceled : BOOL
GET
P_bCanceled := bCanceled;
END_GET
END_PROPERTY

PROPERTY P_bCollFree : BOOL
GET
P_bCollFree := TRUE;
END_GET
END_PROPERTY

PROPERTY P_bError : BOOL
GET
IF eCurrentState = E_MachineState.MACHINESTATE_Error THEN
	P_bError := TRUE;
END_IF
END_GET
END_PROPERTY

PROPERTY P_bHasZSensorSlot : BOOL
GET
END_GET
END_PROPERTY

PROPERTY P_bIsHot : BOOL
GET
END_GET
END_PROPERTY

PROPERTY P_bIsInit : BOOL
GET
END_GET
END_PROPERTY

PROPERTY P_bMeasured : BOOL
GET
P_bMeasured := bMeasured;
END_GET
SET
bMeasured := P_bMeasured;
END_SET
END_PROPERTY

PROPERTY P_bStopAllOnError : BOOL
GET
P_bStopAllOnError := bStopAllOnError;
END_GET
END_PROPERTY

PROPERTY P_bXYIsInit : BOOL
GET
P_bXYIsInit :=  bInitAxisOk AND pXDrive^.P_bHomed AND pYDrive^.P_bHomed;
END_GET
END_PROPERTY

PROPERTY P_bXYIsMoving : BOOL
GET
END_GET
SET
END_SET
END_PROPERTY

PROPERTY P_bZIsMoving : BOOL
GET
END_GET
SET
END_SET
END_PROPERTY

PROPERTY P_eCurrentState : E_MachineState
GET
P_eCurrentState := eCurrentState;
END_GET
SET
END_SET
END_PROPERTY

PROPERTY P_nErrorId : ERRORID
GET
P_nErrorId := stError.ErrorId;
END_GET
END_PROPERTY

PROPERTY P_nNotifyId : UINT
GET
P_nNotifyId := nNotifyId;
END_GET
SET
nNotifyId := P_nNotifyId;
END_SET
END_PROPERTY

PROPERTY P_nNumberOfSlots : UINT
GET
P_nNumberOfSlots := nNumberOfSlots;
END_GET
END_PROPERTY

PROPERTY P_pAssignWorkplate : POINTER TO FB_TargetBase
GET
P_pAssignWorkplate := pAssignWorkplate;
END_GET
END_PROPERTY

PROPERTY P_pFbMultiZ : POINTER TO FB_MultiZRef
GET
P_pFbMultiZ := pFbMultiZ;
END_GET
END_PROPERTY

PROPERTY P_pMzHead : POINTER TO FB_MzHead
GET
END_GET
END_PROPERTY

PROPERTY P_pObject : POINTER TO FB_Object
GET
P_pObject := THIS;
END_GET
END_PROPERTY

